// TwinCAT 3 PLC project kittingDeca
// ProgramVersion: 3.1.4023.0
// libraries:
//   Tc2_DataExchange, * (Beckhoff Automation GmbH)
//   Tc2_EtherCAT, * (Beckhoff Automation GmbH)
//   Tc2_MC2, * (Beckhoff Automation GmbH)
//   Tc2_SerialCom, * (Beckhoff Automation GmbH)
//   Tc2_Standard, * (Beckhoff Automation GmbH)
//   Tc2_System, * (Beckhoff Automation GmbH)
//   Tc2_Utilities, * (Beckhoff Automation GmbH)
//   Tc3_Module, * (Beckhoff Automation GmbH)
//   Tc3_PackML, * (Beckhoff Automation GmbH)
//   VisuDialogs, * (System)
//   VisuSymbols,3.5.10.0,System
// project tree:
//   DUTs/ user_defined_structure.TcDUT (not stored)
//   / GlobalTextList.TcGTLO, PlcTask.TcTTO, VISU_TASK.TcTTO, 视图管理器.TcVMO (not stored)
//   GVLs/ E_DOutputMode.TcDUT (not stored), E_State.TcDUT (not stored), ST_DIO.TcDUT (not stored), ST_IO.TcDUT (not stored), ST_IO_16.TcDUT (not stored), ST_IO_16_int.TcDUT (not stored)
//   GVLs/kitting deca/axis/ AxisHMI_Ex.TcVIS, E_HomingSteps.TcDUT (not stored), FB_MotionAxis_MC.TcPOU, MC_HomeAxis.TcPOU (not stored), ST_MotionAxis_MC.TcDUT
//   GVLs/kitting deca/ DigitalInputStatus.TcDUT (not stored), E_CMD_ConverterMotor.TcDUT, FB_Converter.TcPOU, FB_DigitalInput.TcPOU (not stored), FB_do.TcPOU (not stored), FB_PhotoSensor.TcPOU (not stored), FB_valve.TcPOU, Roller.TcDUT (not stored), Sensor.TcDUT (not stored), ST_Converter.TcDUT, ST_heightDetection.TcDUT, Valve.TcDUT (not stored)
//   GVLs/kitting deca/fixture rotation/ fixtureRotation_Module.TcDUT
//   GVLs/kitting deca/lateral conveyor/ BeltOut.TcDUT, Lateral.TcDUT, LateralBuf_Module.TcDUT, Roller_LC.TcDUT, LateralRecy_Module.TcDUT
//   GVLs/kitting deca/measuring/ ST_byte.TcDUT (not stored), ST_IO_byte.TcDUT (not stored)
//   GVLs/kitting deca/picking module/ Belt.TcDUT, Buffer.TcDUT (not stored), Inner_conveyor.TcDUT, PM_others.TcDUT (not stored), Outter_coveyor.TcDUT (not stored), Picking_Module.TcDUT (not stored), RFID.TcDUT (not stored)
//   GVLs/kitting deca/replenishment module/ arLiftAxis.TcDUT (not stored), Infeed.TcDUT (not stored), Lift.TcDUT (not stored), Outfeed.TcDUT (not stored), Replenishment_Module.TcDUT (not stored)
//   POUs/bagmachines/ AdsArr.TcDUT, BagCmd.TcDUT, BagDetectionCmd.TcDUT, BagDetectionStatus.TcDUT, BagHeightStatus.TcDUT, BagHolderStatus.TcDUT, BagMachineStatus.TcDUT, BagStatus.TcDUT, E_HeightDetection.TcDUT, FB_BagCloser.TcPOU, FB_BagCompactor.TcPOU, FB_BagOpener.TcPOU, fb_interface_bagmachine.TcPOU
//   POUs/ E_RemIndex.TcDUT (not stored), FB_axisCtrl.TcPOU, FB_heightDetection.TcPOU, FB_lbIOmapping.TcPOU, FB_frIOmapping.TcPOU, FB_remAxisMapping.TcPOU, FB_pmAxisMapping.TcPOU, FB_remIOmapping.TcPOU (not stored), FB_lcIOmapping.TcPOU, FB_rmIOmapping.TcPOU, G_HMI.TcGVL, GVL.TcGVL, G_IO.TcGVL, MAIN.TcPOU, ST_axisCtrl.TcDUT (not stored), ST_Color.TcDUT (not stored)
//   VISUs/ OtherList.TcVIS, visu_LC.TcVIS, visu_FR.TcVIS, visu_LB.TcVIS, visu_PM.TcVIS (not stored), visu_Others.TcVIS, visu_ReM.TcVIS, visu_MLC.TcVIS, visu_main.TcVIS, ReMList.TcVIS (not stored), PMList.TcVIS, v_byte.TcVIS (not stored), v_IO_FR.TcVIS, v_IO_fixtureClamp.TcVIS, v_IO_ReM.TcVIS (not stored), v_IO_LC.TcVIS, v_LB.TcVIS, v_rem_0.TcVIS, v_pm_0.TcVIS, v_rem_1.TcVIS
// real-time tasks:
//   TASK PlcTask: cycle T#2ms, priority 12, ADS port 350
//   TASK VISU_TASK: cycle T#200000us, priority 16, ADS port 351
// motion (NC):
//   TASK NC-Task 1 SAF: cycle T#4ms, priority 6, ADS port 501
//   TASK NC-Task 1 SVB: cycle T#10ms, priority 10, ADS port 511
//   AXIS rem0_Lift0 (id 4)
//     Dynamic: Acceleration=15000, Deceleration=15000, Jerk=150000
//     Velo: Maximum=3000
//     OtherSettings: AllowMotionCmdToSlave=true
//     encoder EncType=19
//       EncPara: ScaleFactorNumerator=5, ScaleFactorDenominator=262144, Inverse=true, MaxCount=#xffffffff
//         Inc: RefSoftSyncMask=#x00040000
//     drive DrvType=16
//       DrvPara: Inverse=true, MaxCount=#xffffffff, DriveControlDWord=#x00020100
//         Analog: VeloReferenz=500, TorqueSetpointScale=10, ScaleFactorActTorque=0.1
//         TimeComp: TaskDelayCycles=1
//     controller CtrType=1
//       CtrPara: PriorControlFactor=1
//         PosDiffControl: Range=30
//         Observer: BandWidth=20
//   AXIS rem0_Lift1 (id 5)
//     Dynamic: Acceleration=15000, Deceleration=15000, Jerk=150000
//     Velo: Maximum=3000
//     OtherSettings: AllowMotionCmdToSlave=true
//     encoder EncType=19
//       EncPara: ScaleFactorNumerator=5, ScaleFactorDenominator=262144, Inverse=true, MaxCount=#xffffffff
//         Inc: RefSoftSyncMask=#x00040000
//     drive DrvType=16
//       DrvPara: Inverse=true, MaxCount=#xffffffff, DriveControlDWord=#x00020100
//         Analog: VeloReferenz=500, TorqueSetpointScale=10, ScaleFactorActTorque=0.1
//         TimeComp: TaskDelayCycles=1
//     controller CtrType=1
//       CtrPara: PriorControlFactor=1
//         PosDiffControl: Range=30
//         Observer: BandWidth=20
//   AXIS rem1_Lift0 (id 1)
//     Dynamic: Acceleration=15000, Deceleration=15000, Jerk=150000
//     Velo: Maximum=3000
//     OtherSettings: AllowMotionCmdToSlave=true
//     encoder EncType=19
//       EncPara: ScaleFactorNumerator=5, ScaleFactorDenominator=262144, Inverse=true, MaxCount=#xffffffff
//         Inc: RefSoftSyncMask=#x00040000
//     drive DrvType=16
//       DrvPara: Inverse=true, MaxCount=#xffffffff, DriveControlDWord=#x00020100
//         Analog: VeloReferenz=500, TorqueSetpointScale=10, ScaleFactorActTorque=0.1
//         TimeComp: TaskDelayCycles=1
//     controller CtrType=1
//       CtrPara: PriorControlFactor=1
//         PosDiffControl: Range=30
//         Observer: BandWidth=20
//   AXIS rem1_Lift1 (id 2)
//     Dynamic: Acceleration=15000, Deceleration=15000, Jerk=150000
//     Velo: Maximum=3000
//     OtherSettings: AllowMotionCmdToSlave=true
//     encoder EncType=19
//       EncPara: ScaleFactorNumerator=5, ScaleFactorDenominator=262144, Inverse=true, MaxCount=#xffffffff
//         Inc: RefSoftSyncMask=#x00040000
//     drive DrvType=16
//       DrvPara: Inverse=true, MaxCount=#xffffffff, DriveControlDWord=#x00020100
//         Analog: VeloReferenz=500, TorqueSetpointScale=10, ScaleFactorActTorque=0.1
//         TimeComp: TaskDelayCycles=1
//     controller CtrType=1
//       CtrPara: PriorControlFactor=1
//         PosDiffControl: Range=30
//         Observer: BandWidth=20
//   AXIS rem2_Lift0 (id 9)
//     Dynamic: Acceleration=15000, Deceleration=15000, Jerk=150000
//     Velo: Maximum=3000
//     OtherSettings: AllowMotionCmdToSlave=true
//     encoder EncType=19
//       EncPara: ScaleFactorNumerator=5, ScaleFactorDenominator=262144, Inverse=true, MaxCount=#xffffffff
//         Inc: RefSoftSyncMask=#x00040000
//     drive DrvType=16
//       DrvPara: Inverse=true, MaxCount=#xffffffff, DriveControlDWord=#x00020100
//         Analog: VeloReferenz=500, TorqueSetpointScale=10, ScaleFactorActTorque=0.1
//         TimeComp: TaskDelayCycles=1
//     controller CtrType=1
//       CtrPara: PriorControlFactor=1
//         PosDiffControl: Range=30
//         Observer: BandWidth=20
//   AXIS rem2_Lift1 (id 10)
//     Dynamic: Acceleration=15000, Deceleration=15000, Jerk=150000
//     Velo: Maximum=3000
//     OtherSettings: AllowMotionCmdToSlave=true
//     encoder EncType=19
//       EncPara: ScaleFactorNumerator=5, ScaleFactorDenominator=262144, Inverse=true, MaxCount=#xffffffff
//         Inc: RefSoftSyncMask=#x00040000
//     drive DrvType=16
//       DrvPara: Inverse=true, MaxCount=#xffffffff, DriveControlDWord=#x00020100
//         Analog: VeloReferenz=500, TorqueSetpointScale=10, ScaleFactorActTorque=0.1
//         TimeComp: TaskDelayCycles=1
//     controller CtrType=1
//       CtrPara: PriorControlFactor=1
//         PosDiffControl: Range=30
//         Observer: BandWidth=20
//   AXIS rem3_Lift0 (id 11)
//     Dynamic: Acceleration=15000, Deceleration=15000, Jerk=150000
//     Velo: Maximum=3000
//     OtherSettings: AllowMotionCmdToSlave=true
//     encoder EncType=19
//       EncPara: ScaleFactorNumerator=5, ScaleFactorDenominator=262144, Inverse=true, MaxCount=#xffffffff
//         Inc: RefSoftSyncMask=#x00040000
//     drive DrvType=16
//       DrvPara: Inverse=true, MaxCount=#xffffffff, DriveControlDWord=#x00020100
//         Analog: VeloReferenz=500, TorqueSetpointScale=10, ScaleFactorActTorque=0.1
//         TimeComp: TaskDelayCycles=1
//     controller CtrType=1
//       CtrPara: PriorControlFactor=1
//         PosDiffControl: Range=30
//         Observer: BandWidth=20
//   AXIS rem3_Lift1 (id 12)
//     Dynamic: Acceleration=15000, Deceleration=15000, Jerk=150000
//     Velo: Maximum=3000
//     OtherSettings: AllowMotionCmdToSlave=true
//     encoder EncType=19
//       EncPara: ScaleFactorNumerator=5, ScaleFactorDenominator=262144, Inverse=true, MaxCount=#xffffffff
//         Inc: RefSoftSyncMask=#x00040000
//     drive DrvType=16
//       DrvPara: Inverse=true, MaxCount=#xffffffff, DriveControlDWord=#x00020100
//         Analog: VeloReferenz=500, TorqueSetpointScale=10, ScaleFactorActTorque=0.1
//         TimeComp: TaskDelayCycles=1
//     controller CtrType=1
//       CtrPara: PriorControlFactor=1
//         PosDiffControl: Range=30
//         Observer: BandWidth=20
//   AXIS rem4_Lift0 (id 17)
//     Dynamic: Acceleration=15000, Deceleration=15000, Jerk=150000
//     Velo: Maximum=3000
//     OtherSettings: AllowMotionCmdToSlave=true
//     encoder EncType=19
//       EncPara: ScaleFactorNumerator=5, ScaleFactorDenominator=262144, Inverse=true, MaxCount=#xffffffff
//         Inc: RefSoftSyncMask=#x00040000
//     drive DrvType=16
//       DrvPara: Inverse=true, MaxCount=#xffffffff, DriveControlDWord=#x00020100
//         Analog: VeloReferenz=500, TorqueSetpointScale=10, ScaleFactorActTorque=0.1
//         TimeComp: TaskDelayCycles=1
//     controller CtrType=1
//       CtrPara: PriorControlFactor=1
//         PosDiffControl: Range=30
//         Observer: BandWidth=20
//   AXIS rem4_Lift1 (id 18)
//     Dynamic: Acceleration=15000, Deceleration=15000, Jerk=150000
//     Velo: Maximum=3000
//     OtherSettings: AllowMotionCmdToSlave=true
//     encoder EncType=19
//       EncPara: ScaleFactorNumerator=5, ScaleFactorDenominator=262144, Inverse=true, MaxCount=#xffffffff
//         Inc: RefSoftSyncMask=#x00040000
//     drive DrvType=16
//       DrvPara: Inverse=true, MaxCount=#xffffffff, DriveControlDWord=#x00020100
//         Analog: VeloReferenz=500, TorqueSetpointScale=10, ScaleFactorActTorque=0.1
//         TimeComp: TaskDelayCycles=1
//     controller CtrType=1
//       CtrPara: PriorControlFactor=1
//         PosDiffControl: Range=30
//         Observer: BandWidth=20
//   AXIS rem5_Lift0 (id 19)
//     Dynamic: Acceleration=15000, Deceleration=15000, Jerk=150000
//     Velo: Maximum=3000
//     OtherSettings: AllowMotionCmdToSlave=true
//     encoder EncType=19
//       EncPara: ScaleFactorNumerator=5, ScaleFactorDenominator=262144, Inverse=true, MaxCount=#xffffffff
//         Inc: RefSoftSyncMask=#x00040000
//     drive DrvType=16
//       DrvPara: Inverse=true, MaxCount=#xffffffff, DriveControlDWord=#x00020100
//         Analog: VeloReferenz=500, TorqueSetpointScale=10, ScaleFactorActTorque=0.1
//         TimeComp: TaskDelayCycles=1
//     controller CtrType=1
//       CtrPara: PriorControlFactor=1
//         PosDiffControl: Range=30
//         Observer: BandWidth=20
//   AXIS rem5_Lift1 (id 20)
//     Dynamic: Acceleration=15000, Deceleration=15000, Jerk=150000
//     Velo: Maximum=3000
//     OtherSettings: AllowMotionCmdToSlave=true
//     encoder EncType=19
//       EncPara: ScaleFactorNumerator=5, ScaleFactorDenominator=262144, Inverse=true, MaxCount=#xffffffff
//         Inc: RefSoftSyncMask=#x00040000
//     drive DrvType=16
//       DrvPara: Inverse=true, MaxCount=#xffffffff, DriveControlDWord=#x00020100
//         Analog: VeloReferenz=500, TorqueSetpointScale=10, ScaleFactorActTorque=0.1
//         TimeComp: TaskDelayCycles=1
//     controller CtrType=1
//       CtrPara: PriorControlFactor=1
//         PosDiffControl: Range=30
//         Observer: BandWidth=20
//   AXIS rem6_Lift0 (id 25)
//     Dynamic: Acceleration=15000, Deceleration=15000, Jerk=150000
//     Velo: Maximum=3000
//     OtherSettings: AllowMotionCmdToSlave=true
//     encoder EncType=19
//       EncPara: ScaleFactorNumerator=5, ScaleFactorDenominator=262144, Inverse=true, MaxCount=#xffffffff
//         Inc: RefSoftSyncMask=#x00040000
//     drive DrvType=16
//       DrvPara: Inverse=true, MaxCount=#xffffffff, DriveControlDWord=#x00020100
//         Analog: VeloReferenz=500, TorqueSetpointScale=10, ScaleFactorActTorque=0.1
//         TimeComp: TaskDelayCycles=1
//     controller CtrType=1
//       CtrPara: PriorControlFactor=1
//         PosDiffControl: Range=30
//         Observer: BandWidth=20
//   AXIS rem6_Lift1 (id 26)
//     Dynamic: Acceleration=15000, Deceleration=15000, Jerk=150000
//     Velo: Maximum=3000
//     OtherSettings: AllowMotionCmdToSlave=true
//     encoder EncType=19
//       EncPara: ScaleFactorNumerator=5, ScaleFactorDenominator=262144, Inverse=true, MaxCount=#xffffffff
//         Inc: RefSoftSyncMask=#x00040000
//     drive DrvType=16
//       DrvPara: Inverse=true, MaxCount=#xffffffff, DriveControlDWord=#x00020100
//         Analog: VeloReferenz=500, TorqueSetpointScale=10, ScaleFactorActTorque=0.1
//         TimeComp: TaskDelayCycles=1
//     controller CtrType=1
//       CtrPara: PriorControlFactor=1
//         PosDiffControl: Range=30
//         Observer: BandWidth=20
//   AXIS rem7_Lift0 (id 27)
//     Dynamic: Acceleration=15000, Deceleration=15000, Jerk=150000
//     Velo: Maximum=3000
//     OtherSettings: AllowMotionCmdToSlave=true
//     encoder EncType=19
//       EncPara: ScaleFactorNumerator=5, ScaleFactorDenominator=262144, Inverse=true, MaxCount=#xffffffff
//         Inc: RefSoftSyncMask=#x00040000
//     drive DrvType=16
//       DrvPara: Inverse=true, MaxCount=#xffffffff, DriveControlDWord=#x00020100
//         Analog: VeloReferenz=500, TorqueSetpointScale=10, ScaleFactorActTorque=0.1
//         TimeComp: TaskDelayCycles=1
//     controller CtrType=1
//       CtrPara: PriorControlFactor=1
//         PosDiffControl: Range=30
//         Observer: BandWidth=20
//   AXIS rem7_Lift1 (id 28)
//     Dynamic: Acceleration=15000, Deceleration=15000, Jerk=150000
//     Velo: Maximum=3000
//     OtherSettings: AllowMotionCmdToSlave=true
//     encoder EncType=19
//       EncPara: ScaleFactorNumerator=5, ScaleFactorDenominator=262144, Inverse=true, MaxCount=#xffffffff
//         Inc: RefSoftSyncMask=#x00040000
//     drive DrvType=16
//       DrvPara: Inverse=true, MaxCount=#xffffffff, DriveControlDWord=#x00020100
//         Analog: VeloReferenz=500, TorqueSetpointScale=10, ScaleFactorActTorque=0.1
//         TimeComp: TaskDelayCycles=1
//     controller CtrType=1
//       CtrPara: PriorControlFactor=1
//         PosDiffControl: Range=30
//         Observer: BandWidth=20
//   AXIS rem8_Lift0 (id 33)
//     Dynamic: Acceleration=15000, Deceleration=15000, Jerk=150000
//     Velo: Maximum=3000
//     OtherSettings: AllowMotionCmdToSlave=true
//     encoder EncType=19
//       EncPara: ScaleFactorNumerator=5, ScaleFactorDenominator=262144, Inverse=true, MaxCount=#xffffffff
//         Inc: RefSoftSyncMask=#x00040000
//     drive DrvType=16
//       DrvPara: Inverse=true, MaxCount=#xffffffff, DriveControlDWord=#x00020100
//         Analog: VeloReferenz=500, TorqueSetpointScale=10, ScaleFactorActTorque=0.1
//         TimeComp: TaskDelayCycles=1
//     controller CtrType=1
//       CtrPara: PriorControlFactor=1
//         PosDiffControl: Range=30
//         Observer: BandWidth=20
//   AXIS rem8_Lift1 (id 34)
//     Dynamic: Acceleration=15000, Deceleration=15000, Jerk=150000
//     Velo: Maximum=3000
//     OtherSettings: AllowMotionCmdToSlave=true
//     encoder EncType=19
//       EncPara: ScaleFactorNumerator=5, ScaleFactorDenominator=262144, Inverse=true, MaxCount=#xffffffff
//         Inc: RefSoftSyncMask=#x00040000
//     drive DrvType=16
//       DrvPara: Inverse=true, MaxCount=#xffffffff, DriveControlDWord=#x00020100
//         Analog: VeloReferenz=500, TorqueSetpointScale=10, ScaleFactorActTorque=0.1
//         TimeComp: TaskDelayCycles=1
//     controller CtrType=1
//       CtrPara: PriorControlFactor=1
//         PosDiffControl: Range=30
//         Observer: BandWidth=20
//   AXIS rem9_Lift0 (id 35)
//     Dynamic: Acceleration=15000, Deceleration=15000, Jerk=150000
//     Velo: Maximum=3000
//     OtherSettings: AllowMotionCmdToSlave=true
//     encoder EncType=19
//       EncPara: ScaleFactorNumerator=5, ScaleFactorDenominator=262144, Inverse=true, MaxCount=#xffffffff
//         Inc: RefSoftSyncMask=#x00040000
//     drive DrvType=16
//       DrvPara: Inverse=true, MaxCount=#xffffffff, DriveControlDWord=#x00020100
//         Analog: VeloReferenz=500, TorqueSetpointScale=10, ScaleFactorActTorque=0.1
//         TimeComp: TaskDelayCycles=1
//     controller CtrType=1
//       CtrPara: PriorControlFactor=1
//         PosDiffControl: Range=30
//         Observer: BandWidth=20
//   AXIS rem9_Lift1 (id 36)
//     Dynamic: Acceleration=15000, Deceleration=15000, Jerk=150000
//     Velo: Maximum=3000
//     OtherSettings: AllowMotionCmdToSlave=true
//     encoder EncType=19
//       EncPara: ScaleFactorNumerator=5, ScaleFactorDenominator=262144, Inverse=true, MaxCount=#xffffffff
//         Inc: RefSoftSyncMask=#x00040000
//     drive DrvType=16
//       DrvPara: Inverse=true, MaxCount=#xffffffff, DriveControlDWord=#x00020100
//         Analog: VeloReferenz=500, TorqueSetpointScale=10, ScaleFactorActTorque=0.1
//         TimeComp: TaskDelayCycles=1
//     controller CtrType=1
//       CtrPara: PriorControlFactor=1
//         PosDiffControl: Range=30
//         Observer: BandWidth=20
//   AXIS pm0_buf0 (id 3)
//     Dynamic: Acceleration=15000, Deceleration=15000, Jerk=150000
//     Velo: Maximum=3000
//     OtherSettings: AllowMotionCmdToSlave=true
//     encoder EncType=19
//       EncPara: ScaleFactorNumerator=20.84, ScaleFactorDenominator=262144, MaxCount=#xffffffff
//         Inc: RefSoftSyncMask=#x00040000
//     drive DrvType=16
//       DrvPara: MaxCount=#xffffffff, DriveControlDWord=#x00020100
//         Analog: VeloReferenz=500, TorqueSetpointScale=10, ScaleFactorActTorque=0.1
//         TimeComp: TaskDelayCycles=1
//     controller CtrType=1
//       CtrPara: PriorControlFactor=1
//         PosDiffControl: Range=30
//         Observer: BandWidth=20
//   AXIS pm0_buf1 (id 6)
//     Dynamic: Acceleration=15000, Deceleration=15000, Jerk=150000
//     Velo: Maximum=3000
//     OtherSettings: AllowMotionCmdToSlave=true
//     encoder EncType=19
//       EncPara: ScaleFactorNumerator=20.84, ScaleFactorDenominator=262144, MaxCount=#xffffffff
//         Inc: RefSoftSyncMask=#x00040000
//     drive DrvType=16
//       DrvPara: MaxCount=#xffffffff, DriveControlDWord=#x00020100
//         Analog: VeloReferenz=500, TorqueSetpointScale=10, ScaleFactorActTorque=0.1
//         TimeComp: TaskDelayCycles=1
//     controller CtrType=1
//       CtrPara: PriorControlFactor=1
//         PosDiffControl: Range=30
//         Observer: BandWidth=20
//   AXIS pm1_buf0 (id 7)
//     Dynamic: Acceleration=15000, Deceleration=15000, Jerk=150000
//     Velo: Maximum=3000
//     OtherSettings: AllowMotionCmdToSlave=true
//     encoder EncType=19
//       EncPara: ScaleFactorNumerator=20.84, ScaleFactorDenominator=262144, MaxCount=#xffffffff
//         Inc: RefSoftSyncMask=#x00040000
//     drive DrvType=16
//       DrvPara: MaxCount=#xffffffff, DriveControlDWord=#x00020100
//         Analog: VeloReferenz=500, TorqueSetpointScale=10, ScaleFactorActTorque=0.1
//         TimeComp: TaskDelayCycles=1
//     controller CtrType=1
//       CtrPara: PriorControlFactor=1
//         PosDiffControl: Range=30
//         Observer: BandWidth=20
//   AXIS pm1_buf1 (id 8)
//     Dynamic: Acceleration=15000, Deceleration=15000, Jerk=150000
//     Velo: Maximum=3000
//     OtherSettings: AllowMotionCmdToSlave=true
//     encoder EncType=19
//       EncPara: ScaleFactorNumerator=20.84, ScaleFactorDenominator=262144, MaxCount=#xffffffff
//         Inc: RefSoftSyncMask=#x00040000
//     drive DrvType=16
//       DrvPara: MaxCount=#xffffffff, DriveControlDWord=#x00020100
//         Analog: VeloReferenz=500, TorqueSetpointScale=10, ScaleFactorActTorque=0.1
//         TimeComp: TaskDelayCycles=1
//     controller CtrType=1
//       CtrPara: PriorControlFactor=1
//         PosDiffControl: Range=30
//         Observer: BandWidth=20
//   AXIS pm2_buf0 (id 13)
//     Dynamic: Acceleration=15000, Deceleration=15000, Jerk=150000
//     Velo: Maximum=3000
//     OtherSettings: AllowMotionCmdToSlave=true
//     encoder EncType=19
//       EncPara: ScaleFactorNumerator=20.84, ScaleFactorDenominator=262144, MaxCount=#xffffffff
//         Inc: RefSoftSyncMask=#x00040000
//     drive DrvType=16
//       DrvPara: MaxCount=#xffffffff, DriveControlDWord=#x00020100
//         Analog: VeloReferenz=500, TorqueSetpointScale=10, ScaleFactorActTorque=0.1
//         TimeComp: TaskDelayCycles=1
//     controller CtrType=1
//       CtrPara: PriorControlFactor=1
//         PosDiffControl: Range=30
//         Observer: BandWidth=20
//   AXIS pm2_buf1 (id 14)
//     Dynamic: Acceleration=15000, Deceleration=15000, Jerk=150000
//     Velo: Maximum=3000
//     OtherSettings: AllowMotionCmdToSlave=true
//     encoder EncType=19
//       EncPara: ScaleFactorNumerator=20.84, ScaleFactorDenominator=262144, MaxCount=#xffffffff
//         Inc: RefSoftSyncMask=#x00040000
//     drive DrvType=16
//       DrvPara: MaxCount=#xffffffff, DriveControlDWord=#x00020100
//         Analog: VeloReferenz=500, TorqueSetpointScale=10, ScaleFactorActTorque=0.1
//         TimeComp: TaskDelayCycles=1
//     controller CtrType=1
//       CtrPara: PriorControlFactor=1
//         PosDiffControl: Range=30
//         Observer: BandWidth=20
//   AXIS pm3_buf0 (id 15)
//     Dynamic: Acceleration=15000, Deceleration=15000, Jerk=150000
//     Velo: Maximum=3000
//     OtherSettings: AllowMotionCmdToSlave=true
//     encoder EncType=19
//       EncPara: ScaleFactorNumerator=20.84, ScaleFactorDenominator=262144, MaxCount=#xffffffff
//         Inc: RefSoftSyncMask=#x00040000
//     drive DrvType=16
//       DrvPara: MaxCount=#xffffffff, DriveControlDWord=#x00020100
//         Analog: VeloReferenz=500, TorqueSetpointScale=10, ScaleFactorActTorque=0.1
//         TimeComp: TaskDelayCycles=1
//     controller CtrType=1
//       CtrPara: PriorControlFactor=1
//         PosDiffControl: Range=30
//         Observer: BandWidth=20
//   AXIS pm3_buf1 (id 16)
//     Dynamic: Acceleration=15000, Deceleration=15000, Jerk=150000
//     Velo: Maximum=3000
//     OtherSettings: AllowMotionCmdToSlave=true
//     encoder EncType=19
//       EncPara: ScaleFactorNumerator=20.84, ScaleFactorDenominator=262144, MaxCount=#xffffffff
//         Inc: RefSoftSyncMask=#x00040000
//     drive DrvType=16
//       DrvPara: MaxCount=#xffffffff, DriveControlDWord=#x00020100
//         Analog: VeloReferenz=500, TorqueSetpointScale=10, ScaleFactorActTorque=0.1
//         TimeComp: TaskDelayCycles=1
//     controller CtrType=1
//       CtrPara: PriorControlFactor=1
//         PosDiffControl: Range=30
//         Observer: BandWidth=20
//   AXIS pm4_buf0 (id 21)
//     Dynamic: Acceleration=15000, Deceleration=15000, Jerk=150000
//     Velo: Maximum=3000
//     OtherSettings: AllowMotionCmdToSlave=true
//     encoder EncType=19
//       EncPara: ScaleFactorNumerator=20.84, ScaleFactorDenominator=262144, MaxCount=#xffffffff
//         Inc: RefSoftSyncMask=#x00040000
//     drive DrvType=16
//       DrvPara: MaxCount=#xffffffff, DriveControlDWord=#x00020100
//         Analog: VeloReferenz=500, TorqueSetpointScale=10, ScaleFactorActTorque=0.1
//         TimeComp: TaskDelayCycles=1
//     controller CtrType=1
//       CtrPara: PriorControlFactor=1
//         PosDiffControl: Range=30
//         Observer: BandWidth=20
//   AXIS pm4_buf1 (id 22)
//     Dynamic: Acceleration=15000, Deceleration=15000, Jerk=150000
//     Velo: Maximum=3000
//     OtherSettings: AllowMotionCmdToSlave=true
//     encoder EncType=19
//       EncPara: ScaleFactorNumerator=20.84, ScaleFactorDenominator=262144, MaxCount=#xffffffff
//         Inc: RefSoftSyncMask=#x00040000
//     drive DrvType=16
//       DrvPara: MaxCount=#xffffffff, DriveControlDWord=#x00020100
//         Analog: VeloReferenz=500, TorqueSetpointScale=10, ScaleFactorActTorque=0.1
//         TimeComp: TaskDelayCycles=1
//     controller CtrType=1
//       CtrPara: PriorControlFactor=1
//         PosDiffControl: Range=30
//         Observer: BandWidth=20
//   AXIS pm5_buf0 (id 23)
//     Dynamic: Acceleration=15000, Deceleration=15000, Jerk=150000
//     Velo: Maximum=3000
//     OtherSettings: AllowMotionCmdToSlave=true
//     encoder EncType=19
//       EncPara: ScaleFactorNumerator=20.84, ScaleFactorDenominator=262144, MaxCount=#xffffffff
//         Inc: RefSoftSyncMask=#x00040000
//     drive DrvType=16
//       DrvPara: MaxCount=#xffffffff, DriveControlDWord=#x00020100
//         Analog: VeloReferenz=500, TorqueSetpointScale=10, ScaleFactorActTorque=0.1
//         TimeComp: TaskDelayCycles=1
//     controller CtrType=1
//       CtrPara: PriorControlFactor=1
//         PosDiffControl: Range=30
//         Observer: BandWidth=20
//   AXIS pm5_buf1 (id 24)
//     Dynamic: Acceleration=15000, Deceleration=15000, Jerk=150000
//     Velo: Maximum=3000
//     OtherSettings: AllowMotionCmdToSlave=true
//     encoder EncType=19
//       EncPara: ScaleFactorNumerator=20.84, ScaleFactorDenominator=262144, MaxCount=#xffffffff
//         Inc: RefSoftSyncMask=#x00040000
//     drive DrvType=16
//       DrvPara: MaxCount=#xffffffff, DriveControlDWord=#x00020100
//         Analog: VeloReferenz=500, TorqueSetpointScale=10, ScaleFactorActTorque=0.1
//         TimeComp: TaskDelayCycles=1
//     controller CtrType=1
//       CtrPara: PriorControlFactor=1
//         PosDiffControl: Range=30
//         Observer: BandWidth=20
//   AXIS pm6_buf0 (id 29)
//     Dynamic: Acceleration=15000, Deceleration=15000, Jerk=150000
//     Velo: Maximum=3000
//     OtherSettings: AllowMotionCmdToSlave=true
//     encoder EncType=19
//       EncPara: ScaleFactorNumerator=20.84, ScaleFactorDenominator=262144, MaxCount=#xffffffff
//         Inc: RefSoftSyncMask=#x00040000
//     drive DrvType=16
//       DrvPara: MaxCount=#xffffffff, DriveControlDWord=#x00020100
//         Analog: VeloReferenz=500, TorqueSetpointScale=10, ScaleFactorActTorque=0.1
//         TimeComp: TaskDelayCycles=1
//     controller CtrType=1
//       CtrPara: PriorControlFactor=1
//         PosDiffControl: Range=30
//         Observer: BandWidth=20
//   AXIS pm6_buf1 (id 30)
//     Dynamic: Acceleration=15000, Deceleration=15000, Jerk=150000
//     Velo: Maximum=3000
//     OtherSettings: AllowMotionCmdToSlave=true
//     encoder EncType=19
//       EncPara: ScaleFactorNumerator=20.84, ScaleFactorDenominator=262144, MaxCount=#xffffffff
//         Inc: RefSoftSyncMask=#x00040000
//     drive DrvType=16
//       DrvPara: MaxCount=#xffffffff, DriveControlDWord=#x00020100
//         Analog: VeloReferenz=500, TorqueSetpointScale=10, ScaleFactorActTorque=0.1
//         TimeComp: TaskDelayCycles=1
//     controller CtrType=1
//       CtrPara: PriorControlFactor=1
//         PosDiffControl: Range=30
//         Observer: BandWidth=20
//   AXIS pm7_buf0 (id 31)
//     Dynamic: Acceleration=15000, Deceleration=15000, Jerk=150000
//     Velo: Maximum=3000
//     OtherSettings: AllowMotionCmdToSlave=true
//     encoder EncType=19
//       EncPara: ScaleFactorNumerator=20.84, ScaleFactorDenominator=262144, MaxCount=#xffffffff
//         Inc: RefSoftSyncMask=#x00040000
//     drive DrvType=16
//       DrvPara: MaxCount=#xffffffff, DriveControlDWord=#x00020100
//         Analog: VeloReferenz=500, TorqueSetpointScale=10, ScaleFactorActTorque=0.1
//         TimeComp: TaskDelayCycles=1
//     controller CtrType=1
//       CtrPara: PriorControlFactor=1
//         PosDiffControl: Range=30
//         Observer: BandWidth=20
//   AXIS pm7_buf1 (id 32)
//     Dynamic: Acceleration=15000, Deceleration=15000, Jerk=150000
//     Velo: Maximum=3000
//     OtherSettings: AllowMotionCmdToSlave=true
//     encoder EncType=19
//       EncPara: ScaleFactorNumerator=20.84, ScaleFactorDenominator=262144, MaxCount=#xffffffff
//         Inc: RefSoftSyncMask=#x00040000
//     drive DrvType=16
//       DrvPara: MaxCount=#xffffffff, DriveControlDWord=#x00020100
//         Analog: VeloReferenz=500, TorqueSetpointScale=10, ScaleFactorActTorque=0.1
//         TimeComp: TaskDelayCycles=1
//     controller CtrType=1
//       CtrPara: PriorControlFactor=1
//         PosDiffControl: Range=30
//         Observer: BandWidth=20
//   AXIS pm8_buf0 (id 37)
//     Dynamic: Acceleration=15000, Deceleration=15000, Jerk=150000
//     Velo: Maximum=3000
//     OtherSettings: AllowMotionCmdToSlave=true
//     encoder EncType=19
//       EncPara: ScaleFactorNumerator=20.84, ScaleFactorDenominator=262144, MaxCount=#xffffffff
//         Inc: RefSoftSyncMask=#x00040000
//     drive DrvType=16
//       DrvPara: MaxCount=#xffffffff, DriveControlDWord=#x00020100
//         Analog: VeloReferenz=500, TorqueSetpointScale=10, ScaleFactorActTorque=0.1
//         TimeComp: TaskDelayCycles=1
//     controller CtrType=1
//       CtrPara: PriorControlFactor=1
//         PosDiffControl: Range=30
//         Observer: BandWidth=20
//   AXIS pm8_buf1 (id 38)
//     Dynamic: Acceleration=15000, Deceleration=15000, Jerk=150000
//     Velo: Maximum=3000
//     OtherSettings: AllowMotionCmdToSlave=true
//     encoder EncType=19
//       EncPara: ScaleFactorNumerator=20.84, ScaleFactorDenominator=262144, MaxCount=#xffffffff
//         Inc: RefSoftSyncMask=#x00040000
//     drive DrvType=16
//       DrvPara: MaxCount=#xffffffff, DriveControlDWord=#x00020100
//         Analog: VeloReferenz=500, TorqueSetpointScale=10, ScaleFactorActTorque=0.1
//         TimeComp: TaskDelayCycles=1
//     controller CtrType=1
//       CtrPara: PriorControlFactor=1
//         PosDiffControl: Range=30
//         Observer: BandWidth=20
//   AXIS pm9_buf0 (id 39)
//     Dynamic: Acceleration=15000, Deceleration=15000, Jerk=150000
//     Velo: Maximum=3000
//     OtherSettings: AllowMotionCmdToSlave=true
//     encoder EncType=19
//       EncPara: ScaleFactorNumerator=20.84, ScaleFactorDenominator=262144, MaxCount=#xffffffff
//         Inc: RefSoftSyncMask=#x00040000
//     drive DrvType=16
//       DrvPara: MaxCount=#xffffffff, DriveControlDWord=#x00020100
//         Analog: VeloReferenz=500, TorqueSetpointScale=10, ScaleFactorActTorque=0.1
//         TimeComp: TaskDelayCycles=1
//     controller CtrType=1
//       CtrPara: PriorControlFactor=1
//         PosDiffControl: Range=30
//         Observer: BandWidth=20
//   AXIS pm9_buf1 (id 40)
//     Dynamic: Acceleration=15000, Deceleration=15000, Jerk=150000
//     Velo: Maximum=3000
//     OtherSettings: AllowMotionCmdToSlave=true
//     encoder EncType=19
//       EncPara: ScaleFactorNumerator=20.84, ScaleFactorDenominator=262144, MaxCount=#xffffffff
//         Inc: RefSoftSyncMask=#x00040000
//     drive DrvType=16
//       DrvPara: MaxCount=#xffffffff, DriveControlDWord=#x00020100
//         Analog: VeloReferenz=500, TorqueSetpointScale=10, ScaleFactorActTorque=0.1
//         TimeComp: TaskDelayCycles=1
//     controller CtrType=1
//       CtrPara: PriorControlFactor=1
//         PosDiffControl: Range=30
//         Observer: BandWidth=20
//   AXIS fr0 (id 41)
//     Dynamic: Acceleration=15000, Deceleration=15000, Jerk=150000
//     Velo: Maximum=3000
//     OtherSettings: AllowMotionCmdToSlave=true
//     encoder EncType=19
//       EncPara: ScaleFactorNumerator=7.2, ScaleFactorDenominator=262144, MaxCount=#xffffffff
//         Inc: RefSoftSyncMask=#x00040000
//     drive DrvType=16
//       DrvPara: MaxCount=#xffffffff, DriveControlDWord=#x00020100
//         Analog: VeloReferenz=500, TorqueSetpointScale=10, ScaleFactorActTorque=0.1
//         TimeComp: TaskDelayCycles=1
//     controller CtrType=1
//       CtrPara: PriorControlFactor=1
//         PosDiffControl: Range=30
//         Observer: BandWidth=20
//   AXIS fr1 (id 42)
//     Dynamic: Acceleration=15000, Deceleration=15000, Jerk=150000
//     Velo: Maximum=3000
//     OtherSettings: AllowMotionCmdToSlave=true
//     encoder EncType=19
//       EncPara: ScaleFactorNumerator=7.2, ScaleFactorDenominator=262144, MaxCount=#xffffffff
//         Inc: RefSoftSyncMask=#x00040000
//     drive DrvType=16
//       DrvPara: MaxCount=#xffffffff, DriveControlDWord=#x00020100
//         Analog: VeloReferenz=500, TorqueSetpointScale=10, ScaleFactorActTorque=0.1
//         TimeComp: TaskDelayCycles=1
//     controller CtrType=1
//       CtrPara: PriorControlFactor=1
//         PosDiffControl: Range=30
//         Observer: BandWidth=20
//   AXIS lc0 (id 43)
//     Dynamic: Acceleration=15000, Deceleration=15000, Jerk=150000
//     Velo: Maximum=3000
//     OtherSettings: AllowMotionCmdToSlave=true
//     encoder EncType=19
//       EncPara: ScaleFactorNumerator=20, ScaleFactorDenominator=262144, MaxCount=#xffffffff
//         Inc: RefSoftSyncMask=#x00040000
//     drive DrvType=16
//       DrvPara: MaxCount=#xffffffff, DriveControlDWord=#x00020100
//         Analog: VeloReferenz=1000, TorqueSetpointScale=10, ScaleFactorActTorque=0.1
//         TimeComp: TaskDelayCycles=1
//     controller CtrType=1
//       CtrPara: PriorControlFactor=1
//         PosDiffControl: Range=30
//         Observer: BandWidth=20
//   AXIS lc1 (id 44)
//     Dynamic: Acceleration=15000, Deceleration=15000, Jerk=150000
//     Velo: Maximum=3000
//     OtherSettings: AllowMotionCmdToSlave=true
//     encoder EncType=19
//       EncPara: ScaleFactorNumerator=20, ScaleFactorDenominator=262144, MaxCount=#xffffffff
//         Inc: RefSoftSyncMask=#x00040000
//     drive DrvType=16
//       DrvPara: MaxCount=#xffffffff, DriveControlDWord=#x00020100
//         Analog: VeloReferenz=1000, TorqueSetpointScale=10, ScaleFactorActTorque=0.1
//         TimeComp: TaskDelayCycles=1
//     controller CtrType=1
//       CtrPara: PriorControlFactor=1
//         PosDiffControl: Range=30
//         Observer: BandWidth=20
// I/O:
//   DEVICE Device 1 (EtherCAT Automation Protocol), AmsNetId 192.168.11.159.2.1
//   DEVICE Device 2 (RT-Ethernet Adapter)
//   DEVICE rem_wf, AmsNetId 192.168.11.159.4.1
//     Box 1 (CU2508) [CU2508 Ethernet Port]
//     mcp_dio [GL20-RTU-ECT_1.3.5.0]
//       modules: Module 1 (GL20-1600END), Module 2 (GL20-0016ETP)
//     safetyPLC [Flexi Soft EtherCAT Gateway]
//     rem0_dio [GL20-RTU-ECT_1.3.5.0]
//       modules: DI0, DI1, DI2, DI3, DO0, DO1
//     rem0_Lift0 [SV630_1Axis_03713]
//     rem0_Lift1 [SV630_1Axis_03713]
//     rem0_valve [C2S-EC]
//       modules: Module 1 (C2S-EC-24B)
//     rem1_dio [GL20-RTU-ECT_1.3.5.0]
//       modules: DI4, DI5, DI6, DI7, DO4, DO5
//     rem1_Lift0 [SV630_1Axis_03713]
//     rem1_Lift1 [SV630_1Axis_03713]
//     rem1_valve [C2S-EC]
//       modules: Module 1 (C2S-EC-24B)
//     rem2_dio [GL20-RTU-ECT_1.3.5.0]
//       modules: DI8, DI9, DI10, DI11, DO8, DO9
//     rem2_Lift0 [SV630_1Axis_03713]
//     rem2_Lift1 [SV630_1Axis_03713]
//     rem2_valve [C2S-EC]
//       modules: Module 1 (C2S-EC-24B)
//     rem3_dio [GL20-RTU-ECT_1.3.5.0]
//       modules: DI12, DI13, DI14, DI15, DO12, DO13
//     rem3_Lift0 [SV630_1Axis_03713]
//     rem3_Lift1 [SV630_1Axis_03713]
//     rem3_valve [C2S-EC]
//       modules: Module 1 (C2S-EC-24B)
//     rem4_dio [GL20-RTU-ECT_1.3.5.0]
//       modules: DI0, DI1, DI2, DI3, DO0, DO1
//     rem4_Lift0 [SV630_1Axis_03713]
//     rem4_Lift1 [SV630_1Axis_03713]
//     rem4_valve [C2S-EC]
//       modules: Module 1 (C2S-EC-24B)
//     rem5_dio [GL20-RTU-ECT_1.3.5.0]
//       modules: DI0, DI1, DI2, DI3, DO0, DO1
//     rem5_Lift0 [SV630_1Axis_03713]
//     rem5_Lift1 [SV630_1Axis_03713]
//     rem5_valve [C2S-EC]
//       modules: Module 1 (C2S-EC-24B)
//     rem6_dio [GL20-RTU-ECT_1.3.5.0]
//       modules: DI0, DI1, DI2, DI3, DO0, DO1
//     rem6_Lift0 [SV630_1Axis_03713]
//     rem6_Lift1 [SV630_1Axis_03713]
//     rem6_valve [C2S-EC]
//       modules: Module 1 (C2S-EC-24B)
//     rem7_dio [GL20-RTU-ECT_1.3.5.0]
//       modules: DI0, DI1, DI2, DI3, DO0, DO1
//     rem7_Lift0 [SV630_1Axis_03713]
//     rem7_Lift1 [SV630_1Axis_03713]
//     rem7_valve [C2S-EC]
//       modules: Module 1 (C2S-EC-24B)
//     rem8_dio [GL20-RTU-ECT_1.3.5.0]
//       modules: DI0, DI1, DI2, DI3, DO0, DO1
//     rem8_Lift0 [SV630_1Axis_03713]
//     rem8_Lift1 [SV630_1Axis_03713]
//     rem8_valve [C2S-EC]
//       modules: Module 1 (C2S-EC-24B)
//     rem9_dio [GL20-RTU-ECT_1.3.5.0]
//       modules: DI0, DI1, DI2, DI3, DO0, DO1
//     rem9_Lift0 [SV630_1Axis_03713]
//     rem9_Lift1 [SV630_1Axis_03713]
//     rem9_valve [C2S-EC]
//       modules: Module 1 (C2S-EC-24B)
//     wf4_do [GL20-RTU-ECT_1.3.5.0]
//       modules: Module 1 (GL20-0016ETP), Module 2 (GL20-1600END)
//     wf3_do [GL20-RTU-ECT_1.3.5.0]
//       modules: Module 1 (GL20-0016ETP), Module 2 (GL20-1600END)
//     wf2_do [GL20-RTU-ECT_1.3.5.0]
//       modules: Module 1 (GL20-0016ETP), Module 2 (GL20-1600END)
//     wf1_do [GL20-RTU-ECT_1.3.5.0]
//       modules: Module 1 (GL20-0016ETP), Module 2 (GL20-1600END)
//     wf0_do [GL20-RTU-ECT_1.3.5.0]
//       modules: Module 1 (GL20-0016ETP), Module 2 (GL20-1600END)
//   DEVICE pm side, AmsNetId 192.168.11.159.5.1
//     Box 49 (CU2508) [CU2508 Ethernet Port]
//     lb0_dio [GL20-RTU-ECT_1.3.5.0]
//       modules: Module 1 (GL20-1600END), Module 2 (GL20-0016ETP)
//     lb0_converter [MD800_ECAT_9Axis_V0.19]
//     lc0_dio [GL20-RTU-ECT_1.3.5.0]
//       modules: Module 1 (GL20-1600END), Module 2 (GL20-1600END), Module 3 (GL20-0016ETP), Module 4 (GL20-0016ETP)
//     lc0_converter [MD800_ECAT_9Axis_V0.19]
//     lc0_servermoter [SV630_1Axis_03713]
//     pm0_1_dio [GL20-RTU-ECT_1.3.5.0]
//       modules: Module 1 (GL20-1600END), Module 2 (GL20-1600END), Module 3 (GL20-1600END), Module 4 (GL20-1600END), Module 5 (GL20-1600END), Module 6 (GL20-0016ETP), Module 7 (GL20-0016ETP)
//     pm0_1_innerConv [MD800_ECAT_9Axis_V0.19]
//     pm0_1_outerConv [MD800_ECAT_9Axis_V0.19]
//     pm0_buf0 [SV630_1Axis_03713]
//     pm0_buf1 [SV630_1Axis_03713]
//     pm1_buf0 [SV630_1Axis_03713]
//     pm1_buf1 [SV630_1Axis_03713]
//     pm0_1_RFID [SIG350-0006AP100]
//       modules: Module 1 (IOL_32/32_I/O-Bytes), Module 2 (IOL_32/32_I/O-Bytes), Module 3 (IOL_32/32_I/O-Bytes), Module 4 (IOL_32/32_I/O-Bytes), Module 5 (Slot Empty), Module 6 (Slot Empty), Module 7 (Slot Empty), Module 8 (Slot Empty)
//     fr0_dio [GL20-RTU-ECT_1.3.5.0]
//       modules: Module 1 (GL20-1600END), Module 2 (GL20-0016ETP)
//     fr0_servermotor [SV630_1Axis_03713]
//     pm2_3_dio [GL20-RTU-ECT_1.3.5.0]
//       modules: Module 1 (GL20-1600END), Module 2 (GL20-1600END), Module 3 (GL20-1600END), Module 4 (GL20-1600END), Module 5 (GL20-1600END), Module 6 (GL20-1600END), Module 7 (GL20-0016ETP), Module 8 (GL20-0016ETP)
//     pm2_3_innerConv [MD800_ECAT_9Axis_V0.19]
//     pm2_3_outerConv [MD800_ECAT_9Axis_V0.19]
//     pm2_buf0 [SV630_1Axis_03713]
//     pm2_buf1 [SV630_1Axis_03713]
//     pm3_buf0 [SV630_1Axis_03713]
//     pm3_buf1 [SV630_1Axis_03713]
//     pm2_3_RFID [SIG350-0006AP100]
//       modules: Module 1 (IOL_32/32_I/O-Bytes), Module 2 (IOL_32/32_I/O-Bytes), Module 3 (IOL_32/32_I/O-Bytes), Module 4 (IOL_32/32_I/O-Bytes), Module 5 (Slot Empty), Module 6 (Slot Empty), Module 7 (Slot Empty), Module 8 (Slot Empty)
//     pm4_5_dio [GL20-RTU-ECT_1.3.5.0]
//       modules: Module 1 (GL20-1600END), Module 2 (GL20-1600END), Module 3 (GL20-1600END), Module 4 (GL20-1600END), Module 5 (GL20-1600END), Module 6 (GL20-1600END), Module 7 (GL20-0016ETP), Module 8 (GL20-0016ETP)
//     pm4_5_innerConv [MD800_ECAT_9Axis_V0.19]
//     pm4_5_outerConv [MD800_ECAT_9Axis_V0.19]
//     pm4_buf0 [SV630_1Axis_03713]
//     pm4_buf1 [SV630_1Axis_03713]
//     pm5_buf0 [SV630_1Axis_03713]
//     pm5_buf1 [SV630_1Axis_03713]
//     pm4_5_RFID [SIG350-0006AP100]
//       modules: Module 1 (IOL_32/32_I/O-Bytes), Module 2 (IOL_32/32_I/O-Bytes), Module 3 (IOL_32/32_I/O-Bytes), Module 4 (IOL_32/32_I/O-Bytes), Module 5 (Slot Empty), Module 6 (Slot Empty), Module 7 (Slot Empty), Module 8 (Slot Empty)
//     pm6_7_dio [GL20-RTU-ECT_1.3.5.0]
//       modules: Module 1 (GL20-1600END), Module 2 (GL20-1600END), Module 3 (GL20-1600END), Module 4 (GL20-1600END), Module 5 (GL20-1600END), Module 6 (GL20-0016ETP), Module 7 (GL20-0016ETP)
//     pm6_7_innerConv [MD800_ECAT_9Axis_V0.19]
//     pm6_7_outerConv [MD800_ECAT_9Axis_V0.19]
//     pm6_buf0 [SV630_1Axis_03713]
//     pm6_buf1 [SV630_1Axis_03713]
//     pm7_buf0 [SV630_1Axis_03713]
//     pm7_buf1 [SV630_1Axis_03713]
//     pm6_7_RFID [SIG350-0006AP100]
//       modules: Module 1 (IOL_32/32_I/O-Bytes), Module 2 (IOL_32/32_I/O-Bytes), Module 3 (IOL_32/32_I/O-Bytes), Module 4 (IOL_32/32_I/O-Bytes), Module 5 (Slot Empty), Module 6 (Slot Empty), Module 7 (Slot Empty), Module 8 (Slot Empty)
//     fr1_dio [GL20-RTU-ECT_1.3.5.0]
//       modules: Module 1 (GL20-1600END), Module 2 (GL20-0016ETP)
//     fr1_servermotor [SV630_1Axis_03713]
//     pm8_9_dio [GL20-RTU-ECT_1.3.5.0]
//       modules: Module 1 (GL20-1600END), Module 2 (GL20-1600END), Module 3 (GL20-1600END), Module 4 (GL20-1600END), Module 5 (GL20-1600END), Module 6 (GL20-0016ETP), Module 7 (GL20-0016ETP)
//     pm8_9_innerConv [MD800_ECAT_9Axis_V0.19]
//     pm8_9_outerConv [MD800_ECAT_9Axis_V0.19]
//     pm8_buf0 [SV630_1Axis_03713]
//     pm8_buf1 [SV630_1Axis_03713]
//     pm9_buf0 [SV630_1Axis_03713]
//     pm9_buf1 [SV630_1Axis_03713]
//     pm8_9_RFID [SIG350-0006AP100]
//       modules: Module 1 (IOL_32/32_I/O-Bytes), Module 2 (IOL_32/32_I/O-Bytes), Module 3 (IOL_32/32_I/O-Bytes), Module 4 (IOL_32/32_I/O-Bytes), Module 5 (Slot Empty), Module 6 (Slot Empty), Module 7 (Slot Empty), Module 8 (Slot Empty)
//     lb1_dio [GL20-RTU-ECT_1.3.5.0]
//       modules: Module 1 (GL20-1600END), Module 2 (GL20-0016ETP)
//     lb1_converter [MD800_ECAT_9Axis_V0.19]
//     lc1_dio [GL20-RTU-ECT_1.3.5.0]
//       modules: Module 1 (GL20-1600END), Module 2 (GL20-1600END), Module 3 (GL20-0016ETP), Module 4 (GL20-0016ETP)
//     lc1_converter [MD800_ECAT_9Axis_V0.19]
//     lc1_servermoter [SV630_1Axis_03713]
//   DEVICE Device 5 (USB)
//     Box 1 (CX2100 Power Supply)
//   DEVICE Device 6 (COM Port)
//   DEVICE Device 7 (NOV-DP-RAM)
//   DEVICE Device 8 (EtherCAT) (disabled), AmsNetId 192.168.11.159.9.1
//     Box 63 (DL-EC1A) [DL-EC1A]
// variable links:
//   NC-Task 1 SAF/Axes/fr0 <-> pm side/fr0_servermotor
//     Drive/Inputs/In/nDataIn1 <-> Inputs/Following error actual value
//     Drive/Inputs/In/nDataIn3[0] <-> Inputs/Torque actual value
//     Drive/Inputs/In/nDcOutputTime <-> InfoData/DcOutputShift
//     Drive/Inputs/In/nState1 <-> Inputs/Statusword
//     Drive/Inputs/In/nState2 <-> Inputs/Statusword @bit 8
//     Drive/Inputs/In/nState4 @bit 1 <-> WcState/InputToggle
//     Drive/Inputs/In/nState4 <-> WcState/WcState
//     Drive/Outputs/Out/nCtrl1 <-> Outputs/Controlword
//     Drive/Outputs/Out/nCtrl2 <-> Outputs/Controlword @bit 8
//     Drive/Outputs/Out/nDataOut1 <-> Outputs/Target position
//     Enc/Inputs/In/nDataIn1 <-> Inputs/Position actual value
//     Enc/Inputs/In/nDataIn3 <-> Inputs/Touch probe pos1 pos value
//     Enc/Inputs/In/nDataIn5 <-> Inputs/Touch probe pos2 pos value
//     Enc/Inputs/In/nDcInputTime <-> InfoData/DcInputShift
//     Enc/Inputs/In/nState4 @bit 1 <-> WcState/InputToggle
//     Enc/Inputs/In/nState4 <-> WcState/WcState
//     Enc/Inputs/In/nState5 <-> Inputs/Touch probe status
//     Enc/Inputs/In/nState6 <-> Inputs/Touch probe status @bit 8
//     Enc/Outputs/Out/nCtrl5 <-> Outputs/Touch probe function
//     Enc/Outputs/Out/nCtrl6 <-> Outputs/Touch probe function @bit 8
//   NC-Task 1 SAF/Axes/fr1 <-> pm side/fr1_servermotor
//     Drive/Inputs/In/nDataIn1 <-> Inputs/Following error actual value
//     Drive/Inputs/In/nDataIn3[0] <-> Inputs/Torque actual value
//     Drive/Inputs/In/nDcOutputTime <-> InfoData/DcOutputShift
//     Drive/Inputs/In/nState1 <-> Inputs/Statusword
//     Drive/Inputs/In/nState2 <-> Inputs/Statusword @bit 8
//     Drive/Inputs/In/nState4 @bit 1 <-> WcState/InputToggle
//     Drive/Inputs/In/nState4 <-> WcState/WcState
//     Drive/Outputs/Out/nCtrl1 <-> Outputs/Controlword
//     Drive/Outputs/Out/nCtrl2 <-> Outputs/Controlword @bit 8
//     Drive/Outputs/Out/nDataOut1 <-> Outputs/Target position
//     Enc/Inputs/In/nDataIn1 <-> Inputs/Position actual value
//     Enc/Inputs/In/nDataIn3 <-> Inputs/Touch probe pos1 pos value
//     Enc/Inputs/In/nDataIn5 <-> Inputs/Touch probe pos2 pos value
//     Enc/Inputs/In/nDcInputTime <-> InfoData/DcInputShift
//     Enc/Inputs/In/nState4 @bit 1 <-> WcState/InputToggle
//     Enc/Inputs/In/nState4 <-> WcState/WcState
//     Enc/Inputs/In/nState5 <-> Inputs/Touch probe status
//     Enc/Inputs/In/nState6 <-> Inputs/Touch probe status @bit 8
//     Enc/Outputs/Out/nCtrl5 <-> Outputs/Touch probe function
//     Enc/Outputs/Out/nCtrl6 <-> Outputs/Touch probe function @bit 8
//   NC-Task 1 SAF/Axes/lc0 <-> pm side/lc0_servermoter
//     Drive/Inputs/In/nDataIn1 <-> Inputs/Following error actual value
//     Drive/Inputs/In/nDataIn3[0] <-> Inputs/Torque actual value
//     Drive/Inputs/In/nDcOutputTime <-> InfoData/DcOutputShift
//     Drive/Inputs/In/nState1 <-> Inputs/Statusword
//     Drive/Inputs/In/nState2 <-> Inputs/Statusword @bit 8
//     Drive/Inputs/In/nState4 @bit 1 <-> WcState/InputToggle
//     Drive/Inputs/In/nState4 <-> WcState/WcState
//     Drive/Outputs/Out/nCtrl1 <-> Outputs/Controlword
//     Drive/Outputs/Out/nCtrl2 <-> Outputs/Controlword @bit 8
//     Drive/Outputs/Out/nDataOut1 <-> Outputs/Target position
//     Enc/Inputs/In/nDataIn1 <-> Inputs/Position actual value
//     Enc/Inputs/In/nDataIn3 <-> Inputs/Touch probe pos1 pos value
//     Enc/Inputs/In/nDataIn5 <-> Inputs/Touch probe pos2 pos value
//     Enc/Inputs/In/nDcInputTime <-> InfoData/DcInputShift
//     Enc/Inputs/In/nState4 @bit 1 <-> WcState/InputToggle
//     Enc/Inputs/In/nState4 <-> WcState/WcState
//     Enc/Inputs/In/nState5 <-> Inputs/Touch probe status
//     Enc/Inputs/In/nState6 <-> Inputs/Touch probe status @bit 8
//     Enc/Outputs/Out/nCtrl5 <-> Outputs/Touch probe function
//     Enc/Outputs/Out/nCtrl6 <-> Outputs/Touch probe function @bit 8
//   NC-Task 1 SAF/Axes/lc1 <-> pm side/lc1_servermoter
//     Drive/Inputs/In/nDataIn1 <-> Inputs/Following error actual value
//     Drive/Inputs/In/nDataIn3[0] <-> Inputs/Torque actual value
//     Drive/Inputs/In/nDcOutputTime <-> InfoData/DcOutputShift
//     Drive/Inputs/In/nState1 <-> Inputs/Statusword
//     Drive/Inputs/In/nState2 <-> Inputs/Statusword @bit 8
//     Drive/Inputs/In/nState4 @bit 1 <-> WcState/InputToggle
//     Drive/Inputs/In/nState4 <-> WcState/WcState
//     Drive/Outputs/Out/nCtrl1 <-> Outputs/Controlword
//     Drive/Outputs/Out/nCtrl2 <-> Outputs/Controlword @bit 8
//     Drive/Outputs/Out/nDataOut1 <-> Outputs/Target position
//     Enc/Inputs/In/nDataIn1 <-> Inputs/Position actual value
//     Enc/Inputs/In/nDataIn3 <-> Inputs/Touch probe pos1 pos value
//     Enc/Inputs/In/nDataIn5 <-> Inputs/Touch probe pos2 pos value
//     Enc/Inputs/In/nDcInputTime <-> InfoData/DcInputShift
//     Enc/Inputs/In/nState4 @bit 1 <-> WcState/InputToggle
//     Enc/Inputs/In/nState4 <-> WcState/WcState
//     Enc/Inputs/In/nState5 <-> Inputs/Touch probe status
//     Enc/Inputs/In/nState6 <-> Inputs/Touch probe status @bit 8
//     Enc/Outputs/Out/nCtrl5 <-> Outputs/Touch probe function
//     Enc/Outputs/Out/nCtrl6 <-> Outputs/Touch probe function @bit 8
//   NC-Task 1 SAF/Axes/pm0_buf0 <-> pm side/pm0_buf0
//     Drive/Inputs/In/nDataIn1 <-> Inputs/Following error actual value
//     Drive/Inputs/In/nDataIn3[0] <-> Inputs/Torque actual value
//     Drive/Inputs/In/nDcOutputTime <-> InfoData/DcOutputShift
//     Drive/Inputs/In/nState1 <-> Inputs/Statusword
//     Drive/Inputs/In/nState2 <-> Inputs/Statusword @bit 8
//     Drive/Inputs/In/nState4 @bit 1 <-> WcState/InputToggle
//     Drive/Inputs/In/nState4 <-> WcState/WcState
//     Drive/Outputs/Out/nCtrl1 <-> Outputs/Controlword
//     Drive/Outputs/Out/nCtrl2 <-> Outputs/Controlword @bit 8
//     Drive/Outputs/Out/nDataOut1 <-> Outputs/Target position
//     Enc/Inputs/In/nDataIn1 <-> Inputs/Position actual value
//     Enc/Inputs/In/nDataIn3 <-> Inputs/Touch probe pos1 pos value
//     Enc/Inputs/In/nDataIn5 <-> Inputs/Touch probe pos2 pos value
//     Enc/Inputs/In/nDcInputTime <-> InfoData/DcInputShift
//     Enc/Inputs/In/nState4 @bit 1 <-> WcState/InputToggle
//     Enc/Inputs/In/nState4 <-> WcState/WcState
//     Enc/Inputs/In/nState5 <-> Inputs/Touch probe status
//     Enc/Inputs/In/nState6 <-> Inputs/Touch probe status @bit 8
//     Enc/Outputs/Out/nCtrl5 <-> Outputs/Touch probe function
//     Enc/Outputs/Out/nCtrl6 <-> Outputs/Touch probe function @bit 8
//   NC-Task 1 SAF/Axes/pm0_buf1 <-> pm side/pm0_buf1
//     Drive/Inputs/In/nDataIn1 <-> Inputs/Following error actual value
//     Drive/Inputs/In/nDataIn3[0] <-> Inputs/Torque actual value
//     Drive/Inputs/In/nDcOutputTime <-> InfoData/DcOutputShift
//     Drive/Inputs/In/nState1 <-> Inputs/Statusword
//     Drive/Inputs/In/nState2 <-> Inputs/Statusword @bit 8
//     Drive/Inputs/In/nState4 @bit 1 <-> WcState/InputToggle
//     Drive/Inputs/In/nState4 <-> WcState/WcState
//     Drive/Outputs/Out/nCtrl1 <-> Outputs/Controlword
//     Drive/Outputs/Out/nCtrl2 <-> Outputs/Controlword @bit 8
//     Drive/Outputs/Out/nDataOut1 <-> Outputs/Target position
//     Enc/Inputs/In/nDataIn1 <-> Inputs/Position actual value
//     Enc/Inputs/In/nDataIn3 <-> Inputs/Touch probe pos1 pos value
//     Enc/Inputs/In/nDataIn5 <-> Inputs/Touch probe pos2 pos value
//     Enc/Inputs/In/nDcInputTime <-> InfoData/DcInputShift
//     Enc/Inputs/In/nState4 @bit 1 <-> WcState/InputToggle
//     Enc/Inputs/In/nState4 <-> WcState/WcState
//     Enc/Inputs/In/nState5 <-> Inputs/Touch probe status
//     Enc/Inputs/In/nState6 <-> Inputs/Touch probe status @bit 8
//     Enc/Outputs/Out/nCtrl5 <-> Outputs/Touch probe function
//     Enc/Outputs/Out/nCtrl6 <-> Outputs/Touch probe function @bit 8
//   NC-Task 1 SAF/Axes/pm1_buf0 <-> pm side/pm1_buf0
//     Drive/Inputs/In/nDataIn1 <-> Inputs/Following error actual value
//     Drive/Inputs/In/nDataIn3[0] <-> Inputs/Torque actual value
//     Drive/Inputs/In/nDcOutputTime <-> InfoData/DcOutputShift
//     Drive/Inputs/In/nState1 <-> Inputs/Statusword
//     Drive/Inputs/In/nState2 <-> Inputs/Statusword @bit 8
//     Drive/Inputs/In/nState4 @bit 1 <-> WcState/InputToggle
//     Drive/Inputs/In/nState4 <-> WcState/WcState
//     Drive/Outputs/Out/nCtrl1 <-> Outputs/Controlword
//     Drive/Outputs/Out/nCtrl2 <-> Outputs/Controlword @bit 8
//     Drive/Outputs/Out/nDataOut1 <-> Outputs/Target position
//     Enc/Inputs/In/nDataIn1 <-> Inputs/Position actual value
//     Enc/Inputs/In/nDataIn3 <-> Inputs/Touch probe pos1 pos value
//     Enc/Inputs/In/nDataIn5 <-> Inputs/Touch probe pos2 pos value
//     Enc/Inputs/In/nDcInputTime <-> InfoData/DcInputShift
//     Enc/Inputs/In/nState4 @bit 1 <-> WcState/InputToggle
//     Enc/Inputs/In/nState4 <-> WcState/WcState
//     Enc/Inputs/In/nState5 <-> Inputs/Touch probe status
//     Enc/Inputs/In/nState6 <-> Inputs/Touch probe status @bit 8
//     Enc/Outputs/Out/nCtrl5 <-> Outputs/Touch probe function
//     Enc/Outputs/Out/nCtrl6 <-> Outputs/Touch probe function @bit 8
//   NC-Task 1 SAF/Axes/pm1_buf1 <-> pm side/pm1_buf1
//     Drive/Inputs/In/nDataIn1 <-> Inputs/Following error actual value
//     Drive/Inputs/In/nDataIn3[0] <-> Inputs/Torque actual value
//     Drive/Inputs/In/nDcOutputTime <-> InfoData/DcOutputShift
//     Drive/Inputs/In/nState1 <-> Inputs/Statusword
//     Drive/Inputs/In/nState2 <-> Inputs/Statusword @bit 8
//     Drive/Inputs/In/nState4 @bit 1 <-> WcState/InputToggle
//     Drive/Inputs/In/nState4 <-> WcState/WcState
//     Drive/Outputs/Out/nCtrl1 <-> Outputs/Controlword
//     Drive/Outputs/Out/nCtrl2 <-> Outputs/Controlword @bit 8
//     Drive/Outputs/Out/nDataOut1 <-> Outputs/Target position
//     Enc/Inputs/In/nDataIn1 <-> Inputs/Position actual value
//     Enc/Inputs/In/nDataIn3 <-> Inputs/Touch probe pos1 pos value
//     Enc/Inputs/In/nDataIn5 <-> Inputs/Touch probe pos2 pos value
//     Enc/Inputs/In/nDcInputTime <-> InfoData/DcInputShift
//     Enc/Inputs/In/nState4 @bit 1 <-> WcState/InputToggle
//     Enc/Inputs/In/nState4 <-> WcState/WcState
//     Enc/Inputs/In/nState5 <-> Inputs/Touch probe status
//     Enc/Inputs/In/nState6 <-> Inputs/Touch probe status @bit 8
//     Enc/Outputs/Out/nCtrl5 <-> Outputs/Touch probe function
//     Enc/Outputs/Out/nCtrl6 <-> Outputs/Touch probe function @bit 8
//   NC-Task 1 SAF/Axes/pm2_buf0 <-> pm side/pm2_buf0
//     Drive/Inputs/In/nDataIn1 <-> Inputs/Following error actual value
//     Drive/Inputs/In/nDataIn3[0] <-> Inputs/Torque actual value
//     Drive/Inputs/In/nDcOutputTime <-> InfoData/DcOutputShift
//     Drive/Inputs/In/nState1 <-> Inputs/Statusword
//     Drive/Inputs/In/nState2 <-> Inputs/Statusword @bit 8
//     Drive/Inputs/In/nState4 @bit 1 <-> WcState/InputToggle
//     Drive/Inputs/In/nState4 <-> WcState/WcState
//     Drive/Outputs/Out/nCtrl1 <-> Outputs/Controlword
//     Drive/Outputs/Out/nCtrl2 <-> Outputs/Controlword @bit 8
//     Drive/Outputs/Out/nDataOut1 <-> Outputs/Target position
//     Enc/Inputs/In/nDataIn1 <-> Inputs/Position actual value
//     Enc/Inputs/In/nDataIn3 <-> Inputs/Touch probe pos1 pos value
//     Enc/Inputs/In/nDataIn5 <-> Inputs/Touch probe pos2 pos value
//     Enc/Inputs/In/nDcInputTime <-> InfoData/DcInputShift
//     Enc/Inputs/In/nState4 @bit 1 <-> WcState/InputToggle
//     Enc/Inputs/In/nState4 <-> WcState/WcState
//     Enc/Inputs/In/nState5 <-> Inputs/Touch probe status
//     Enc/Inputs/In/nState6 <-> Inputs/Touch probe status @bit 8
//     Enc/Outputs/Out/nCtrl5 <-> Outputs/Touch probe function
//     Enc/Outputs/Out/nCtrl6 <-> Outputs/Touch probe function @bit 8
//   NC-Task 1 SAF/Axes/pm2_buf1 <-> pm side/pm2_buf1
//     Drive/Inputs/In/nDataIn1 <-> Inputs/Following error actual value
//     Drive/Inputs/In/nDataIn3[0] <-> Inputs/Torque actual value
//     Drive/Inputs/In/nDcOutputTime <-> InfoData/DcOutputShift
//     Drive/Inputs/In/nState1 <-> Inputs/Statusword
//     Drive/Inputs/In/nState2 <-> Inputs/Statusword @bit 8
//     Drive/Inputs/In/nState4 @bit 1 <-> WcState/InputToggle
//     Drive/Inputs/In/nState4 <-> WcState/WcState
//     Drive/Outputs/Out/nCtrl1 <-> Outputs/Controlword
//     Drive/Outputs/Out/nCtrl2 <-> Outputs/Controlword @bit 8
//     Drive/Outputs/Out/nDataOut1 <-> Outputs/Target position
//     Enc/Inputs/In/nDataIn1 <-> Inputs/Position actual value
//     Enc/Inputs/In/nDataIn3 <-> Inputs/Touch probe pos1 pos value
//     Enc/Inputs/In/nDataIn5 <-> Inputs/Touch probe pos2 pos value
//     Enc/Inputs/In/nDcInputTime <-> InfoData/DcInputShift
//     Enc/Inputs/In/nState4 @bit 1 <-> WcState/InputToggle
//     Enc/Inputs/In/nState4 <-> WcState/WcState
//     Enc/Inputs/In/nState5 <-> Inputs/Touch probe status
//     Enc/Inputs/In/nState6 <-> Inputs/Touch probe status @bit 8
//     Enc/Outputs/Out/nCtrl5 <-> Outputs/Touch probe function
//     Enc/Outputs/Out/nCtrl6 <-> Outputs/Touch probe function @bit 8
//   NC-Task 1 SAF/Axes/pm3_buf0 <-> pm side/pm3_buf0
//     Drive/Inputs/In/nDataIn1 <-> Inputs/Following error actual value
//     Drive/Inputs/In/nDataIn3[0] <-> Inputs/Torque actual value
//     Drive/Inputs/In/nDcOutputTime <-> InfoData/DcOutputShift
//     Drive/Inputs/In/nState1 <-> Inputs/Statusword
//     Drive/Inputs/In/nState2 <-> Inputs/Statusword @bit 8
//     Drive/Inputs/In/nState4 @bit 1 <-> WcState/InputToggle
//     Drive/Inputs/In/nState4 <-> WcState/WcState
//     Drive/Outputs/Out/nCtrl1 <-> Outputs/Controlword
//     Drive/Outputs/Out/nCtrl2 <-> Outputs/Controlword @bit 8
//     Drive/Outputs/Out/nDataOut1 <-> Outputs/Target position
//     Enc/Inputs/In/nDataIn1 <-> Inputs/Position actual value
//     Enc/Inputs/In/nDataIn3 <-> Inputs/Touch probe pos1 pos value
//     Enc/Inputs/In/nDataIn5 <-> Inputs/Touch probe pos2 pos value
//     Enc/Inputs/In/nDcInputTime <-> InfoData/DcInputShift
//     Enc/Inputs/In/nState4 @bit 1 <-> WcState/InputToggle
//     Enc/Inputs/In/nState4 <-> WcState/WcState
//     Enc/Inputs/In/nState5 <-> Inputs/Touch probe status
//     Enc/Inputs/In/nState6 <-> Inputs/Touch probe status @bit 8
//     Enc/Outputs/Out/nCtrl5 <-> Outputs/Touch probe function
//     Enc/Outputs/Out/nCtrl6 <-> Outputs/Touch probe function @bit 8
//   NC-Task 1 SAF/Axes/pm3_buf1 <-> pm side/pm3_buf1
//     Drive/Inputs/In/nDataIn1 <-> Inputs/Following error actual value
//     Drive/Inputs/In/nDataIn3[0] <-> Inputs/Torque actual value
//     Drive/Inputs/In/nDcOutputTime <-> InfoData/DcOutputShift
//     Drive/Inputs/In/nState1 <-> Inputs/Statusword
//     Drive/Inputs/In/nState2 <-> Inputs/Statusword @bit 8
//     Drive/Inputs/In/nState4 @bit 1 <-> WcState/InputToggle
//     Drive/Inputs/In/nState4 <-> WcState/WcState
//     Drive/Outputs/Out/nCtrl1 <-> Outputs/Controlword
//     Drive/Outputs/Out/nCtrl2 <-> Outputs/Controlword @bit 8
//     Drive/Outputs/Out/nDataOut1 <-> Outputs/Target position
//     Enc/Inputs/In/nDataIn1 <-> Inputs/Position actual value
//     Enc/Inputs/In/nDataIn3 <-> Inputs/Touch probe pos1 pos value
//     Enc/Inputs/In/nDataIn5 <-> Inputs/Touch probe pos2 pos value
//     Enc/Inputs/In/nDcInputTime <-> InfoData/DcInputShift
//     Enc/Inputs/In/nState4 @bit 1 <-> WcState/InputToggle
//     Enc/Inputs/In/nState4 <-> WcState/WcState
//     Enc/Inputs/In/nState5 <-> Inputs/Touch probe status
//     Enc/Inputs/In/nState6 <-> Inputs/Touch probe status @bit 8
//     Enc/Outputs/Out/nCtrl5 <-> Outputs/Touch probe function
//     Enc/Outputs/Out/nCtrl6 <-> Outputs/Touch probe function @bit 8
//   NC-Task 1 SAF/Axes/pm4_buf0 <-> pm side/pm4_buf0
//     Drive/Inputs/In/nDataIn1 <-> Inputs/Following error actual value
//     Drive/Inputs/In/nDataIn3[0] <-> Inputs/Torque actual value
//     Drive/Inputs/In/nDcOutputTime <-> InfoData/DcOutputShift
//     Drive/Inputs/In/nState1 <-> Inputs/Statusword
//     Drive/Inputs/In/nState2 <-> Inputs/Statusword @bit 8
//     Drive/Inputs/In/nState4 @bit 1 <-> WcState/InputToggle
//     Drive/Inputs/In/nState4 <-> WcState/WcState
//     Drive/Outputs/Out/nCtrl1 <-> Outputs/Controlword
//     Drive/Outputs/Out/nCtrl2 <-> Outputs/Controlword @bit 8
//     Drive/Outputs/Out/nDataOut1 <-> Outputs/Target position
//     Enc/Inputs/In/nDataIn1 <-> Inputs/Position actual value
//     Enc/Inputs/In/nDataIn3 <-> Inputs/Touch probe pos1 pos value
//     Enc/Inputs/In/nDataIn5 <-> Inputs/Touch probe pos2 pos value
//     Enc/Inputs/In/nDcInputTime <-> InfoData/DcInputShift
//     Enc/Inputs/In/nState4 @bit 1 <-> WcState/InputToggle
//     Enc/Inputs/In/nState4 <-> WcState/WcState
//     Enc/Inputs/In/nState5 <-> Inputs/Touch probe status
//     Enc/Inputs/In/nState6 <-> Inputs/Touch probe status @bit 8
//     Enc/Outputs/Out/nCtrl5 <-> Outputs/Touch probe function
//     Enc/Outputs/Out/nCtrl6 <-> Outputs/Touch probe function @bit 8
//   NC-Task 1 SAF/Axes/pm4_buf1 <-> pm side/pm4_buf1
//     Drive/Inputs/In/nDataIn1 <-> Inputs/Following error actual value
//     Drive/Inputs/In/nDataIn3[0] <-> Inputs/Torque actual value
//     Drive/Inputs/In/nDcOutputTime <-> InfoData/DcOutputShift
//     Drive/Inputs/In/nState1 <-> Inputs/Statusword
//     Drive/Inputs/In/nState2 <-> Inputs/Statusword @bit 8
//     Drive/Inputs/In/nState4 @bit 1 <-> WcState/InputToggle
//     Drive/Inputs/In/nState4 <-> WcState/WcState
//     Drive/Outputs/Out/nCtrl1 <-> Outputs/Controlword
//     Drive/Outputs/Out/nCtrl2 <-> Outputs/Controlword @bit 8
//     Drive/Outputs/Out/nDataOut1 <-> Outputs/Target position
//     Enc/Inputs/In/nDataIn1 <-> Inputs/Position actual value
//     Enc/Inputs/In/nDataIn3 <-> Inputs/Touch probe pos1 pos value
//     Enc/Inputs/In/nDataIn5 <-> Inputs/Touch probe pos2 pos value
//     Enc/Inputs/In/nDcInputTime <-> InfoData/DcInputShift
//     Enc/Inputs/In/nState4 @bit 1 <-> WcState/InputToggle
//     Enc/Inputs/In/nState4 <-> WcState/WcState
//     Enc/Inputs/In/nState5 <-> Inputs/Touch probe status
//     Enc/Inputs/In/nState6 <-> Inputs/Touch probe status @bit 8
//     Enc/Outputs/Out/nCtrl5 <-> Outputs/Touch probe function
//     Enc/Outputs/Out/nCtrl6 <-> Outputs/Touch probe function @bit 8
//   NC-Task 1 SAF/Axes/pm5_buf0 <-> pm side/pm5_buf0
//     Drive/Inputs/In/nDataIn1 <-> Inputs/Following error actual value
//     Drive/Inputs/In/nDataIn3[0] <-> Inputs/Torque actual value
//     Drive/Inputs/In/nDcOutputTime <-> InfoData/DcOutputShift
//     Drive/Inputs/In/nState1 <-> Inputs/Statusword
//     Drive/Inputs/In/nState2 <-> Inputs/Statusword @bit 8
//     Drive/Inputs/In/nState4 @bit 1 <-> WcState/InputToggle
//     Drive/Inputs/In/nState4 <-> WcState/WcState
//     Drive/Outputs/Out/nCtrl1 <-> Outputs/Controlword
//     Drive/Outputs/Out/nCtrl2 <-> Outputs/Controlword @bit 8
//     Drive/Outputs/Out/nDataOut1 <-> Outputs/Target position
//     Enc/Inputs/In/nDataIn1 <-> Inputs/Position actual value
//     Enc/Inputs/In/nDataIn3 <-> Inputs/Touch probe pos1 pos value
//     Enc/Inputs/In/nDataIn5 <-> Inputs/Touch probe pos2 pos value
//     Enc/Inputs/In/nDcInputTime <-> InfoData/DcInputShift
//     Enc/Inputs/In/nState4 @bit 1 <-> WcState/InputToggle
//     Enc/Inputs/In/nState4 <-> WcState/WcState
//     Enc/Inputs/In/nState5 <-> Inputs/Touch probe status
//     Enc/Inputs/In/nState6 <-> Inputs/Touch probe status @bit 8
//     Enc/Outputs/Out/nCtrl5 <-> Outputs/Touch probe function
//     Enc/Outputs/Out/nCtrl6 <-> Outputs/Touch probe function @bit 8
//   NC-Task 1 SAF/Axes/pm5_buf1 <-> pm side/pm5_buf1
//     Drive/Inputs/In/nDataIn1 <-> Inputs/Following error actual value
//     Drive/Inputs/In/nDataIn3[0] <-> Inputs/Torque actual value
//     Drive/Inputs/In/nDcOutputTime <-> InfoData/DcOutputShift
//     Drive/Inputs/In/nState1 <-> Inputs/Statusword
//     Drive/Inputs/In/nState2 <-> Inputs/Statusword @bit 8
//     Drive/Inputs/In/nState4 @bit 1 <-> WcState/InputToggle
//     Drive/Inputs/In/nState4 <-> WcState/WcState
//     Drive/Outputs/Out/nCtrl1 <-> Outputs/Controlword
//     Drive/Outputs/Out/nCtrl2 <-> Outputs/Controlword @bit 8
//     Drive/Outputs/Out/nDataOut1 <-> Outputs/Target position
//     Enc/Inputs/In/nDataIn1 <-> Inputs/Position actual value
//     Enc/Inputs/In/nDataIn3 <-> Inputs/Touch probe pos1 pos value
//     Enc/Inputs/In/nDataIn5 <-> Inputs/Touch probe pos2 pos value
//     Enc/Inputs/In/nDcInputTime <-> InfoData/DcInputShift
//     Enc/Inputs/In/nState4 @bit 1 <-> WcState/InputToggle
//     Enc/Inputs/In/nState4 <-> WcState/WcState
//     Enc/Inputs/In/nState5 <-> Inputs/Touch probe status
//     Enc/Inputs/In/nState6 <-> Inputs/Touch probe status @bit 8
//     Enc/Outputs/Out/nCtrl5 <-> Outputs/Touch probe function
//     Enc/Outputs/Out/nCtrl6 <-> Outputs/Touch probe function @bit 8
//   NC-Task 1 SAF/Axes/pm6_buf0 <-> pm side/pm6_buf0
//     Drive/Inputs/In/nDataIn1 <-> Inputs/Following error actual value
//     Drive/Inputs/In/nDataIn3[0] <-> Inputs/Torque actual value
//     Drive/Inputs/In/nDcOutputTime <-> InfoData/DcOutputShift
//     Drive/Inputs/In/nState1 <-> Inputs/Statusword
//     Drive/Inputs/In/nState2 <-> Inputs/Statusword @bit 8
//     Drive/Inputs/In/nState4 @bit 1 <-> WcState/InputToggle
//     Drive/Inputs/In/nState4 <-> WcState/WcState
//     Drive/Outputs/Out/nCtrl1 <-> Outputs/Controlword
//     Drive/Outputs/Out/nCtrl2 <-> Outputs/Controlword @bit 8
//     Drive/Outputs/Out/nDataOut1 <-> Outputs/Target position
//     Enc/Inputs/In/nDataIn1 <-> Inputs/Position actual value
//     Enc/Inputs/In/nDataIn3 <-> Inputs/Touch probe pos1 pos value
//     Enc/Inputs/In/nDataIn5 <-> Inputs/Touch probe pos2 pos value
//     Enc/Inputs/In/nDcInputTime <-> InfoData/DcInputShift
//     Enc/Inputs/In/nState4 @bit 1 <-> WcState/InputToggle
//     Enc/Inputs/In/nState4 <-> WcState/WcState
//     Enc/Inputs/In/nState5 <-> Inputs/Touch probe status
//     Enc/Inputs/In/nState6 <-> Inputs/Touch probe status @bit 8
//     Enc/Outputs/Out/nCtrl5 <-> Outputs/Touch probe function
//     Enc/Outputs/Out/nCtrl6 <-> Outputs/Touch probe function @bit 8
//   NC-Task 1 SAF/Axes/pm6_buf1 <-> pm side/pm6_buf1
//     Drive/Inputs/In/nDataIn1 <-> Inputs/Following error actual value
//     Drive/Inputs/In/nDataIn3[0] <-> Inputs/Torque actual value
//     Drive/Inputs/In/nDcOutputTime <-> InfoData/DcOutputShift
//     Drive/Inputs/In/nState1 <-> Inputs/Statusword
//     Drive/Inputs/In/nState2 <-> Inputs/Statusword @bit 8
//     Drive/Inputs/In/nState4 @bit 1 <-> WcState/InputToggle
//     Drive/Inputs/In/nState4 <-> WcState/WcState
//     Drive/Outputs/Out/nCtrl1 <-> Outputs/Controlword
//     Drive/Outputs/Out/nCtrl2 <-> Outputs/Controlword @bit 8
//     Drive/Outputs/Out/nDataOut1 <-> Outputs/Target position
//     Enc/Inputs/In/nDataIn1 <-> Inputs/Position actual value
//     Enc/Inputs/In/nDataIn3 <-> Inputs/Touch probe pos1 pos value
//     Enc/Inputs/In/nDataIn5 <-> Inputs/Touch probe pos2 pos value
//     Enc/Inputs/In/nDcInputTime <-> InfoData/DcInputShift
//     Enc/Inputs/In/nState4 @bit 1 <-> WcState/InputToggle
//     Enc/Inputs/In/nState4 <-> WcState/WcState
//     Enc/Inputs/In/nState5 <-> Inputs/Touch probe status
//     Enc/Inputs/In/nState6 <-> Inputs/Touch probe status @bit 8
//     Enc/Outputs/Out/nCtrl5 <-> Outputs/Touch probe function
//     Enc/Outputs/Out/nCtrl6 <-> Outputs/Touch probe function @bit 8
//   NC-Task 1 SAF/Axes/pm7_buf0 <-> pm side/pm7_buf0
//     Drive/Inputs/In/nDataIn1 <-> Inputs/Following error actual value
//     Drive/Inputs/In/nDataIn3[0] <-> Inputs/Torque actual value
//     Drive/Inputs/In/nDcOutputTime <-> InfoData/DcOutputShift
//     Drive/Inputs/In/nState1 <-> Inputs/Statusword
//     Drive/Inputs/In/nState2 <-> Inputs/Statusword @bit 8
//     Drive/Inputs/In/nState4 @bit 1 <-> WcState/InputToggle
//     Drive/Inputs/In/nState4 <-> WcState/WcState
//     Drive/Outputs/Out/nCtrl1 <-> Outputs/Controlword
//     Drive/Outputs/Out/nCtrl2 <-> Outputs/Controlword @bit 8
//     Drive/Outputs/Out/nDataOut1 <-> Outputs/Target position
//     Enc/Inputs/In/nDataIn1 <-> Inputs/Position actual value
//     Enc/Inputs/In/nDataIn3 <-> Inputs/Touch probe pos1 pos value
//     Enc/Inputs/In/nDataIn5 <-> Inputs/Touch probe pos2 pos value
//     Enc/Inputs/In/nDcInputTime <-> InfoData/DcInputShift
//     Enc/Inputs/In/nState4 @bit 1 <-> WcState/InputToggle
//     Enc/Inputs/In/nState4 <-> WcState/WcState
//     Enc/Inputs/In/nState5 <-> Inputs/Touch probe status
//     Enc/Inputs/In/nState6 <-> Inputs/Touch probe status @bit 8
//     Enc/Outputs/Out/nCtrl5 <-> Outputs/Touch probe function
//     Enc/Outputs/Out/nCtrl6 <-> Outputs/Touch probe function @bit 8
//   NC-Task 1 SAF/Axes/pm7_buf1 <-> pm side/pm7_buf1
//     Drive/Inputs/In/nDataIn1 <-> Inputs/Following error actual value
//     Drive/Inputs/In/nDataIn3[0] <-> Inputs/Torque actual value
//     Drive/Inputs/In/nDcOutputTime <-> InfoData/DcOutputShift
//     Drive/Inputs/In/nState1 <-> Inputs/Statusword
//     Drive/Inputs/In/nState2 <-> Inputs/Statusword @bit 8
//     Drive/Inputs/In/nState4 @bit 1 <-> WcState/InputToggle
//     Drive/Inputs/In/nState4 <-> WcState/WcState
//     Drive/Outputs/Out/nCtrl1 <-> Outputs/Controlword
//     Drive/Outputs/Out/nCtrl2 <-> Outputs/Controlword @bit 8
//     Drive/Outputs/Out/nDataOut1 <-> Outputs/Target position
//     Enc/Inputs/In/nDataIn1 <-> Inputs/Position actual value
//     Enc/Inputs/In/nDataIn3 <-> Inputs/Touch probe pos1 pos value
//     Enc/Inputs/In/nDataIn5 <-> Inputs/Touch probe pos2 pos value
//     Enc/Inputs/In/nDcInputTime <-> InfoData/DcInputShift
//     Enc/Inputs/In/nState4 @bit 1 <-> WcState/InputToggle
//     Enc/Inputs/In/nState4 <-> WcState/WcState
//     Enc/Inputs/In/nState5 <-> Inputs/Touch probe status
//     Enc/Inputs/In/nState6 <-> Inputs/Touch probe status @bit 8
//     Enc/Outputs/Out/nCtrl5 <-> Outputs/Touch probe function
//     Enc/Outputs/Out/nCtrl6 <-> Outputs/Touch probe function @bit 8
//   NC-Task 1 SAF/Axes/pm8_buf0 <-> pm side/pm8_buf0
//     Drive/Inputs/In/nDataIn1 <-> Inputs/Following error actual value
//     Drive/Inputs/In/nDataIn3[0] <-> Inputs/Torque actual value
//     Drive/Inputs/In/nDcOutputTime <-> InfoData/DcOutputShift
//     Drive/Inputs/In/nState1 <-> Inputs/Statusword
//     Drive/Inputs/In/nState2 <-> Inputs/Statusword @bit 8
//     Drive/Inputs/In/nState4 @bit 1 <-> WcState/InputToggle
//     Drive/Inputs/In/nState4 <-> WcState/WcState
//     Drive/Outputs/Out/nCtrl1 <-> Outputs/Controlword
//     Drive/Outputs/Out/nCtrl2 <-> Outputs/Controlword @bit 8
//     Drive/Outputs/Out/nDataOut1 <-> Outputs/Target position
//     Enc/Inputs/In/nDataIn1 <-> Inputs/Position actual value
//     Enc/Inputs/In/nDataIn3 <-> Inputs/Touch probe pos1 pos value
//     Enc/Inputs/In/nDataIn5 <-> Inputs/Touch probe pos2 pos value
//     Enc/Inputs/In/nDcInputTime <-> InfoData/DcInputShift
//     Enc/Inputs/In/nState4 @bit 1 <-> WcState/InputToggle
//     Enc/Inputs/In/nState4 <-> WcState/WcState
//     Enc/Inputs/In/nState5 <-> Inputs/Touch probe status
//     Enc/Inputs/In/nState6 <-> Inputs/Touch probe status @bit 8
//     Enc/Outputs/Out/nCtrl5 <-> Outputs/Touch probe function
//     Enc/Outputs/Out/nCtrl6 <-> Outputs/Touch probe function @bit 8
//   NC-Task 1 SAF/Axes/pm8_buf1 <-> pm side/pm8_buf1
//     Drive/Inputs/In/nDataIn1 <-> Inputs/Following error actual value
//     Drive/Inputs/In/nDataIn3[0] <-> Inputs/Torque actual value
//     Drive/Inputs/In/nDcOutputTime <-> InfoData/DcOutputShift
//     Drive/Inputs/In/nState1 <-> Inputs/Statusword
//     Drive/Inputs/In/nState2 <-> Inputs/Statusword @bit 8
//     Drive/Inputs/In/nState4 @bit 1 <-> WcState/InputToggle
//     Drive/Inputs/In/nState4 <-> WcState/WcState
//     Drive/Outputs/Out/nCtrl1 <-> Outputs/Controlword
//     Drive/Outputs/Out/nCtrl2 <-> Outputs/Controlword @bit 8
//     Drive/Outputs/Out/nDataOut1 <-> Outputs/Target position
//     Enc/Inputs/In/nDataIn1 <-> Inputs/Position actual value
//     Enc/Inputs/In/nDataIn3 <-> Inputs/Touch probe pos1 pos value
//     Enc/Inputs/In/nDataIn5 <-> Inputs/Touch probe pos2 pos value
//     Enc/Inputs/In/nDcInputTime <-> InfoData/DcInputShift
//     Enc/Inputs/In/nState4 @bit 1 <-> WcState/InputToggle
//     Enc/Inputs/In/nState4 <-> WcState/WcState
//     Enc/Inputs/In/nState5 <-> Inputs/Touch probe status
//     Enc/Inputs/In/nState6 <-> Inputs/Touch probe status @bit 8
//     Enc/Outputs/Out/nCtrl5 <-> Outputs/Touch probe function
//     Enc/Outputs/Out/nCtrl6 <-> Outputs/Touch probe function @bit 8
//   NC-Task 1 SAF/Axes/pm9_buf0 <-> pm side/pm9_buf0
//     Drive/Inputs/In/nDataIn1 <-> Inputs/Following error actual value
//     Drive/Inputs/In/nDataIn3[0] <-> Inputs/Torque actual value
//     Drive/Inputs/In/nDcOutputTime <-> InfoData/DcOutputShift
//     Drive/Inputs/In/nState1 <-> Inputs/Statusword
//     Drive/Inputs/In/nState2 <-> Inputs/Statusword @bit 8
//     Drive/Inputs/In/nState4 @bit 1 <-> WcState/InputToggle
//     Drive/Inputs/In/nState4 <-> WcState/WcState
//     Drive/Outputs/Out/nCtrl1 <-> Outputs/Controlword
//     Drive/Outputs/Out/nCtrl2 <-> Outputs/Controlword @bit 8
//     Drive/Outputs/Out/nDataOut1 <-> Outputs/Target position
//     Enc/Inputs/In/nDataIn1 <-> Inputs/Position actual value
//     Enc/Inputs/In/nDataIn3 <-> Inputs/Touch probe pos1 pos value
//     Enc/Inputs/In/nDataIn5 <-> Inputs/Touch probe pos2 pos value
//     Enc/Inputs/In/nDcInputTime <-> InfoData/DcInputShift
//     Enc/Inputs/In/nState4 @bit 1 <-> WcState/InputToggle
//     Enc/Inputs/In/nState4 <-> WcState/WcState
//     Enc/Inputs/In/nState5 <-> Inputs/Touch probe status
//     Enc/Inputs/In/nState6 <-> Inputs/Touch probe status @bit 8
//     Enc/Outputs/Out/nCtrl5 <-> Outputs/Touch probe function
//     Enc/Outputs/Out/nCtrl6 <-> Outputs/Touch probe function @bit 8
//   NC-Task 1 SAF/Axes/pm9_buf1 <-> pm side/pm9_buf1
//     Drive/Inputs/In/nDataIn1 <-> Inputs/Following error actual value
//     Drive/Inputs/In/nDataIn3[0] <-> Inputs/Torque actual value
//     Drive/Inputs/In/nDcOutputTime <-> InfoData/DcOutputShift
//     Drive/Inputs/In/nState1 <-> Inputs/Statusword
//     Drive/Inputs/In/nState2 <-> Inputs/Statusword @bit 8
//     Drive/Inputs/In/nState4 @bit 1 <-> WcState/InputToggle
//     Drive/Inputs/In/nState4 <-> WcState/WcState
//     Drive/Outputs/Out/nCtrl1 <-> Outputs/Controlword
//     Drive/Outputs/Out/nCtrl2 <-> Outputs/Controlword @bit 8
//     Drive/Outputs/Out/nDataOut1 <-> Outputs/Target position
//     Enc/Inputs/In/nDataIn1 <-> Inputs/Position actual value
//     Enc/Inputs/In/nDataIn3 <-> Inputs/Touch probe pos1 pos value
//     Enc/Inputs/In/nDataIn5 <-> Inputs/Touch probe pos2 pos value
//     Enc/Inputs/In/nDcInputTime <-> InfoData/DcInputShift
//     Enc/Inputs/In/nState4 @bit 1 <-> WcState/InputToggle
//     Enc/Inputs/In/nState4 <-> WcState/WcState
//     Enc/Inputs/In/nState5 <-> Inputs/Touch probe status
//     Enc/Inputs/In/nState6 <-> Inputs/Touch probe status @bit 8
//     Enc/Outputs/Out/nCtrl5 <-> Outputs/Touch probe function
//     Enc/Outputs/Out/nCtrl6 <-> Outputs/Touch probe function @bit 8
//   NC-Task 1 SAF/Axes/rem0_Lift0 <-> rem_wf/rem0_Lift0
//     Drive/Inputs/In/nDataIn1 <-> Inputs/Following error actual value
//     Drive/Inputs/In/nDataIn3[0] <-> Inputs/Torque actual value
//     Drive/Inputs/In/nDcOutputTime <-> InfoData/DcOutputShift
//     Drive/Inputs/In/nState1 <-> Inputs/Statusword
//     Drive/Inputs/In/nState2 <-> Inputs/Statusword @bit 8
//     Drive/Inputs/In/nState4 @bit 1 <-> WcState/InputToggle
//     Drive/Inputs/In/nState4 <-> WcState/WcState
//     Drive/Outputs/Out/nCtrl1 <-> Outputs/Controlword
//     Drive/Outputs/Out/nCtrl2 <-> Outputs/Controlword @bit 8
//     Drive/Outputs/Out/nDataOut1 <-> Outputs/Target position
//     Enc/Inputs/In/nDataIn1 <-> Inputs/Position actual value
//     Enc/Inputs/In/nDataIn3 <-> Inputs/Touch probe pos1 pos value
//     Enc/Inputs/In/nDataIn5 <-> Inputs/Touch probe pos2 pos value
//     Enc/Inputs/In/nDcInputTime <-> InfoData/DcInputShift
//     Enc/Inputs/In/nState4 @bit 1 <-> WcState/InputToggle
//     Enc/Inputs/In/nState4 <-> WcState/WcState
//     Enc/Inputs/In/nState5 <-> Inputs/Touch probe status
//     Enc/Inputs/In/nState6 <-> Inputs/Touch probe status @bit 8
//     Enc/Outputs/Out/nCtrl5 <-> Outputs/Touch probe function
//     Enc/Outputs/Out/nCtrl6 <-> Outputs/Touch probe function @bit 8
//   NC-Task 1 SAF/Axes/rem0_Lift1 <-> rem_wf/rem0_Lift1
//     Drive/Inputs/In/nDataIn1 <-> Inputs/Following error actual value
//     Drive/Inputs/In/nDataIn3[0] <-> Inputs/Torque actual value
//     Drive/Inputs/In/nDcOutputTime <-> InfoData/DcOutputShift
//     Drive/Inputs/In/nState1 <-> Inputs/Statusword
//     Drive/Inputs/In/nState2 <-> Inputs/Statusword @bit 8
//     Drive/Inputs/In/nState4 @bit 1 <-> WcState/InputToggle
//     Drive/Inputs/In/nState4 <-> WcState/WcState
//     Drive/Outputs/Out/nCtrl1 <-> Outputs/Controlword
//     Drive/Outputs/Out/nCtrl2 <-> Outputs/Controlword @bit 8
//     Drive/Outputs/Out/nDataOut1 <-> Outputs/Target position
//     Enc/Inputs/In/nDataIn1 <-> Inputs/Position actual value
//     Enc/Inputs/In/nDataIn3 <-> Inputs/Touch probe pos1 pos value
//     Enc/Inputs/In/nDataIn5 <-> Inputs/Touch probe pos2 pos value
//     Enc/Inputs/In/nDcInputTime <-> InfoData/DcInputShift
//     Enc/Inputs/In/nState4 @bit 1 <-> WcState/InputToggle
//     Enc/Inputs/In/nState4 <-> WcState/WcState
//     Enc/Inputs/In/nState5 <-> Inputs/Touch probe status
//     Enc/Inputs/In/nState6 <-> Inputs/Touch probe status @bit 8
//     Enc/Outputs/Out/nCtrl5 <-> Outputs/Touch probe function
//     Enc/Outputs/Out/nCtrl6 <-> Outputs/Touch probe function @bit 8
//   NC-Task 1 SAF/Axes/rem1_Lift0 <-> rem_wf/rem1_Lift0
//     Drive/Inputs/In/nDataIn1 <-> Inputs/Following error actual value
//     Drive/Inputs/In/nDataIn3[0] <-> Inputs/Torque actual value
//     Drive/Inputs/In/nDcOutputTime <-> InfoData/DcOutputShift
//     Drive/Inputs/In/nState1 <-> Inputs/Statusword
//     Drive/Inputs/In/nState2 <-> Inputs/Statusword @bit 8
//     Drive/Inputs/In/nState4 @bit 1 <-> WcState/InputToggle
//     Drive/Inputs/In/nState4 <-> WcState/WcState
//     Drive/Outputs/Out/nCtrl1 <-> Outputs/Controlword
//     Drive/Outputs/Out/nCtrl2 <-> Outputs/Controlword @bit 8
//     Drive/Outputs/Out/nDataOut1 <-> Outputs/Target position
//     Enc/Inputs/In/nDataIn1 <-> Inputs/Position actual value
//     Enc/Inputs/In/nDataIn3 <-> Inputs/Touch probe pos1 pos value
//     Enc/Inputs/In/nDataIn5 <-> Inputs/Touch probe pos2 pos value
//     Enc/Inputs/In/nDcInputTime <-> InfoData/DcInputShift
//     Enc/Inputs/In/nState4 @bit 1 <-> WcState/InputToggle
//     Enc/Inputs/In/nState4 <-> WcState/WcState
//     Enc/Inputs/In/nState5 <-> Inputs/Touch probe status
//     Enc/Inputs/In/nState6 <-> Inputs/Touch probe status @bit 8
//     Enc/Outputs/Out/nCtrl5 <-> Outputs/Touch probe function
//     Enc/Outputs/Out/nCtrl6 <-> Outputs/Touch probe function @bit 8
//   NC-Task 1 SAF/Axes/rem1_Lift1 <-> rem_wf/rem1_Lift1
//     Drive/Inputs/In/nDataIn1 <-> Inputs/Following error actual value
//     Drive/Inputs/In/nDataIn3[0] <-> Inputs/Torque actual value
//     Drive/Inputs/In/nDcOutputTime <-> InfoData/DcOutputShift
//     Drive/Inputs/In/nState1 <-> Inputs/Statusword
//     Drive/Inputs/In/nState2 <-> Inputs/Statusword @bit 8
//     Drive/Inputs/In/nState4 @bit 1 <-> WcState/InputToggle
//     Drive/Inputs/In/nState4 <-> WcState/WcState
//     Drive/Outputs/Out/nCtrl1 <-> Outputs/Controlword
//     Drive/Outputs/Out/nCtrl2 <-> Outputs/Controlword @bit 8
//     Drive/Outputs/Out/nDataOut1 <-> Outputs/Target position
//     Enc/Inputs/In/nDataIn1 <-> Inputs/Position actual value
//     Enc/Inputs/In/nDataIn3 <-> Inputs/Touch probe pos1 pos value
//     Enc/Inputs/In/nDataIn5 <-> Inputs/Touch probe pos2 pos value
//     Enc/Inputs/In/nDcInputTime <-> InfoData/DcInputShift
//     Enc/Inputs/In/nState4 @bit 1 <-> WcState/InputToggle
//     Enc/Inputs/In/nState4 <-> WcState/WcState
//     Enc/Inputs/In/nState5 <-> Inputs/Touch probe status
//     Enc/Inputs/In/nState6 <-> Inputs/Touch probe status @bit 8
//     Enc/Outputs/Out/nCtrl5 <-> Outputs/Touch probe function
//     Enc/Outputs/Out/nCtrl6 <-> Outputs/Touch probe function @bit 8
//   NC-Task 1 SAF/Axes/rem2_Lift0 <-> rem_wf/rem2_Lift0
//     Drive/Inputs/In/nDataIn1 <-> Inputs/Following error actual value
//     Drive/Inputs/In/nDataIn3[0] <-> Inputs/Torque actual value
//     Drive/Inputs/In/nDcOutputTime <-> InfoData/DcOutputShift
//     Drive/Inputs/In/nState1 <-> Inputs/Statusword
//     Drive/Inputs/In/nState2 <-> Inputs/Statusword @bit 8
//     Drive/Inputs/In/nState4 @bit 1 <-> WcState/InputToggle
//     Drive/Inputs/In/nState4 <-> WcState/WcState
//     Drive/Outputs/Out/nCtrl1 <-> Outputs/Controlword
//     Drive/Outputs/Out/nCtrl2 <-> Outputs/Controlword @bit 8
//     Drive/Outputs/Out/nDataOut1 <-> Outputs/Target position
//     Enc/Inputs/In/nDataIn1 <-> Inputs/Position actual value
//     Enc/Inputs/In/nDataIn3 <-> Inputs/Touch probe pos1 pos value
//     Enc/Inputs/In/nDataIn5 <-> Inputs/Touch probe pos2 pos value
//     Enc/Inputs/In/nDcInputTime <-> InfoData/DcInputShift
//     Enc/Inputs/In/nState4 @bit 1 <-> WcState/InputToggle
//     Enc/Inputs/In/nState4 <-> WcState/WcState
//     Enc/Inputs/In/nState5 <-> Inputs/Touch probe status
//     Enc/Inputs/In/nState6 <-> Inputs/Touch probe status @bit 8
//     Enc/Outputs/Out/nCtrl5 <-> Outputs/Touch probe function
//     Enc/Outputs/Out/nCtrl6 <-> Outputs/Touch probe function @bit 8
//   NC-Task 1 SAF/Axes/rem2_Lift1 <-> rem_wf/rem2_Lift1
//     Drive/Inputs/In/nDataIn1 <-> Inputs/Following error actual value
//     Drive/Inputs/In/nDataIn3[0] <-> Inputs/Torque actual value
//     Drive/Inputs/In/nDcOutputTime <-> InfoData/DcOutputShift
//     Drive/Inputs/In/nState1 <-> Inputs/Statusword
//     Drive/Inputs/In/nState2 <-> Inputs/Statusword @bit 8
//     Drive/Inputs/In/nState4 @bit 1 <-> WcState/InputToggle
//     Drive/Inputs/In/nState4 <-> WcState/WcState
//     Drive/Outputs/Out/nCtrl1 <-> Outputs/Controlword
//     Drive/Outputs/Out/nCtrl2 <-> Outputs/Controlword @bit 8
//     Drive/Outputs/Out/nDataOut1 <-> Outputs/Target position
//     Enc/Inputs/In/nDataIn1 <-> Inputs/Position actual value
//     Enc/Inputs/In/nDataIn3 <-> Inputs/Touch probe pos1 pos value
//     Enc/Inputs/In/nDataIn5 <-> Inputs/Touch probe pos2 pos value
//     Enc/Inputs/In/nDcInputTime <-> InfoData/DcInputShift
//     Enc/Inputs/In/nState4 @bit 1 <-> WcState/InputToggle
//     Enc/Inputs/In/nState4 <-> WcState/WcState
//     Enc/Inputs/In/nState5 <-> Inputs/Touch probe status
//     Enc/Inputs/In/nState6 <-> Inputs/Touch probe status @bit 8
//     Enc/Outputs/Out/nCtrl5 <-> Outputs/Touch probe function
//     Enc/Outputs/Out/nCtrl6 <-> Outputs/Touch probe function @bit 8
//   NC-Task 1 SAF/Axes/rem3_Lift0 <-> rem_wf/rem3_Lift0
//     Drive/Inputs/In/nDataIn1 <-> Inputs/Following error actual value
//     Drive/Inputs/In/nDataIn3[0] <-> Inputs/Torque actual value
//     Drive/Inputs/In/nDcOutputTime <-> InfoData/DcOutputShift
//     Drive/Inputs/In/nState1 <-> Inputs/Statusword
//     Drive/Inputs/In/nState2 <-> Inputs/Statusword @bit 8
//     Drive/Inputs/In/nState4 @bit 1 <-> WcState/InputToggle
//     Drive/Inputs/In/nState4 <-> WcState/WcState
//     Drive/Outputs/Out/nCtrl1 <-> Outputs/Controlword
//     Drive/Outputs/Out/nCtrl2 <-> Outputs/Controlword @bit 8
//     Drive/Outputs/Out/nDataOut1 <-> Outputs/Target position
//     Enc/Inputs/In/nDataIn1 <-> Inputs/Position actual value
//     Enc/Inputs/In/nDataIn3 <-> Inputs/Touch probe pos1 pos value
//     Enc/Inputs/In/nDataIn5 <-> Inputs/Touch probe pos2 pos value
//     Enc/Inputs/In/nDcInputTime <-> InfoData/DcInputShift
//     Enc/Inputs/In/nState4 @bit 1 <-> WcState/InputToggle
//     Enc/Inputs/In/nState4 <-> WcState/WcState
//     Enc/Inputs/In/nState5 <-> Inputs/Touch probe status
//     Enc/Inputs/In/nState6 <-> Inputs/Touch probe status @bit 8
//     Enc/Outputs/Out/nCtrl5 <-> Outputs/Touch probe function
//     Enc/Outputs/Out/nCtrl6 <-> Outputs/Touch probe function @bit 8
//   NC-Task 1 SAF/Axes/rem3_Lift1 <-> rem_wf/rem3_Lift1
//     Drive/Inputs/In/nDataIn1 <-> Inputs/Following error actual value
//     Drive/Inputs/In/nDataIn3[0] <-> Inputs/Torque actual value
//     Drive/Inputs/In/nDcOutputTime <-> InfoData/DcOutputShift
//     Drive/Inputs/In/nState1 <-> Inputs/Statusword
//     Drive/Inputs/In/nState2 <-> Inputs/Statusword @bit 8
//     Drive/Inputs/In/nState4 @bit 1 <-> WcState/InputToggle
//     Drive/Inputs/In/nState4 <-> WcState/WcState
//     Drive/Outputs/Out/nCtrl1 <-> Outputs/Controlword
//     Drive/Outputs/Out/nCtrl2 <-> Outputs/Controlword @bit 8
//     Drive/Outputs/Out/nDataOut1 <-> Outputs/Target position
//     Enc/Inputs/In/nDataIn1 <-> Inputs/Position actual value
//     Enc/Inputs/In/nDataIn3 <-> Inputs/Touch probe pos1 pos value
//     Enc/Inputs/In/nDataIn5 <-> Inputs/Touch probe pos2 pos value
//     Enc/Inputs/In/nDcInputTime <-> InfoData/DcInputShift
//     Enc/Inputs/In/nState4 @bit 1 <-> WcState/InputToggle
//     Enc/Inputs/In/nState4 <-> WcState/WcState
//     Enc/Inputs/In/nState5 <-> Inputs/Touch probe status
//     Enc/Inputs/In/nState6 <-> Inputs/Touch probe status @bit 8
//     Enc/Outputs/Out/nCtrl5 <-> Outputs/Touch probe function
//     Enc/Outputs/Out/nCtrl6 <-> Outputs/Touch probe function @bit 8
//   NC-Task 1 SAF/Axes/rem4_Lift0 <-> rem_wf/rem4_Lift0
//     Drive/Inputs/In/nDataIn1 <-> Inputs/Following error actual value
//     Drive/Inputs/In/nDataIn3[0] <-> Inputs/Torque actual value
//     Drive/Inputs/In/nDcOutputTime <-> InfoData/DcOutputShift
//     Drive/Inputs/In/nState1 <-> Inputs/Statusword
//     Drive/Inputs/In/nState2 <-> Inputs/Statusword @bit 8
//     Drive/Inputs/In/nState4 @bit 1 <-> WcState/InputToggle
//     Drive/Inputs/In/nState4 <-> WcState/WcState
//     Drive/Outputs/Out/nCtrl1 <-> Outputs/Controlword
//     Drive/Outputs/Out/nCtrl2 <-> Outputs/Controlword @bit 8
//     Drive/Outputs/Out/nDataOut1 <-> Outputs/Target position
//     Enc/Inputs/In/nDataIn1 <-> Inputs/Position actual value
//     Enc/Inputs/In/nDataIn3 <-> Inputs/Touch probe pos1 pos value
//     Enc/Inputs/In/nDataIn5 <-> Inputs/Touch probe pos2 pos value
//     Enc/Inputs/In/nDcInputTime <-> InfoData/DcInputShift
//     Enc/Inputs/In/nState4 @bit 1 <-> WcState/InputToggle
//     Enc/Inputs/In/nState4 <-> WcState/WcState
//     Enc/Inputs/In/nState5 <-> Inputs/Touch probe status
//     Enc/Inputs/In/nState6 <-> Inputs/Touch probe status @bit 8
//     Enc/Outputs/Out/nCtrl5 <-> Outputs/Touch probe function
//     Enc/Outputs/Out/nCtrl6 <-> Outputs/Touch probe function @bit 8
//   NC-Task 1 SAF/Axes/rem4_Lift1 <-> rem_wf/rem4_Lift1
//     Drive/Inputs/In/nDataIn1 <-> Inputs/Following error actual value
//     Drive/Inputs/In/nDataIn3[0] <-> Inputs/Torque actual value
//     Drive/Inputs/In/nDcOutputTime <-> InfoData/DcOutputShift
//     Drive/Inputs/In/nState1 <-> Inputs/Statusword
//     Drive/Inputs/In/nState2 <-> Inputs/Statusword @bit 8
//     Drive/Inputs/In/nState4 @bit 1 <-> WcState/InputToggle
//     Drive/Inputs/In/nState4 <-> WcState/WcState
//     Drive/Outputs/Out/nCtrl1 <-> Outputs/Controlword
//     Drive/Outputs/Out/nCtrl2 <-> Outputs/Controlword @bit 8
//     Drive/Outputs/Out/nDataOut1 <-> Outputs/Target position
//     Enc/Inputs/In/nDataIn1 <-> Inputs/Position actual value
//     Enc/Inputs/In/nDataIn3 <-> Inputs/Touch probe pos1 pos value
//     Enc/Inputs/In/nDataIn5 <-> Inputs/Touch probe pos2 pos value
//     Enc/Inputs/In/nDcInputTime <-> InfoData/DcInputShift
//     Enc/Inputs/In/nState4 @bit 1 <-> WcState/InputToggle
//     Enc/Inputs/In/nState4 <-> WcState/WcState
//     Enc/Inputs/In/nState5 <-> Inputs/Touch probe status
//     Enc/Inputs/In/nState6 <-> Inputs/Touch probe status @bit 8
//     Enc/Outputs/Out/nCtrl5 <-> Outputs/Touch probe function
//     Enc/Outputs/Out/nCtrl6 <-> Outputs/Touch probe function @bit 8
//   NC-Task 1 SAF/Axes/rem5_Lift0 <-> rem_wf/rem5_Lift0
//     Drive/Inputs/In/nDataIn1 <-> Inputs/Following error actual value
//     Drive/Inputs/In/nDataIn3[0] <-> Inputs/Torque actual value
//     Drive/Inputs/In/nDcOutputTime <-> InfoData/DcOutputShift
//     Drive/Inputs/In/nState1 <-> Inputs/Statusword
//     Drive/Inputs/In/nState2 <-> Inputs/Statusword @bit 8
//     Drive/Inputs/In/nState4 @bit 1 <-> WcState/InputToggle
//     Drive/Inputs/In/nState4 <-> WcState/WcState
//     Drive/Outputs/Out/nCtrl1 <-> Outputs/Controlword
//     Drive/Outputs/Out/nCtrl2 <-> Outputs/Controlword @bit 8
//     Drive/Outputs/Out/nDataOut1 <-> Outputs/Target position
//     Enc/Inputs/In/nDataIn1 <-> Inputs/Position actual value
//     Enc/Inputs/In/nDataIn3 <-> Inputs/Touch probe pos1 pos value
//     Enc/Inputs/In/nDataIn5 <-> Inputs/Touch probe pos2 pos value
//     Enc/Inputs/In/nDcInputTime <-> InfoData/DcInputShift
//     Enc/Inputs/In/nState4 @bit 1 <-> WcState/InputToggle
//     Enc/Inputs/In/nState4 <-> WcState/WcState
//     Enc/Inputs/In/nState5 <-> Inputs/Touch probe status
//     Enc/Inputs/In/nState6 <-> Inputs/Touch probe status @bit 8
//     Enc/Outputs/Out/nCtrl5 <-> Outputs/Touch probe function
//     Enc/Outputs/Out/nCtrl6 <-> Outputs/Touch probe function @bit 8
//   NC-Task 1 SAF/Axes/rem5_Lift1 <-> rem_wf/rem5_Lift1
//     Drive/Inputs/In/nDataIn1 <-> Inputs/Following error actual value
//     Drive/Inputs/In/nDataIn3[0] <-> Inputs/Torque actual value
//     Drive/Inputs/In/nDcOutputTime <-> InfoData/DcOutputShift
//     Drive/Inputs/In/nState1 <-> Inputs/Statusword
//     Drive/Inputs/In/nState2 <-> Inputs/Statusword @bit 8
//     Drive/Inputs/In/nState4 @bit 1 <-> WcState/InputToggle
//     Drive/Inputs/In/nState4 <-> WcState/WcState
//     Drive/Outputs/Out/nCtrl1 <-> Outputs/Controlword
//     Drive/Outputs/Out/nCtrl2 <-> Outputs/Controlword @bit 8
//     Drive/Outputs/Out/nDataOut1 <-> Outputs/Target position
//     Enc/Inputs/In/nDataIn1 <-> Inputs/Position actual value
//     Enc/Inputs/In/nDataIn3 <-> Inputs/Touch probe pos1 pos value
//     Enc/Inputs/In/nDataIn5 <-> Inputs/Touch probe pos2 pos value
//     Enc/Inputs/In/nDcInputTime <-> InfoData/DcInputShift
//     Enc/Inputs/In/nState4 @bit 1 <-> WcState/InputToggle
//     Enc/Inputs/In/nState4 <-> WcState/WcState
//     Enc/Inputs/In/nState5 <-> Inputs/Touch probe status
//     Enc/Inputs/In/nState6 <-> Inputs/Touch probe status @bit 8
//     Enc/Outputs/Out/nCtrl5 <-> Outputs/Touch probe function
//     Enc/Outputs/Out/nCtrl6 <-> Outputs/Touch probe function @bit 8
//   NC-Task 1 SAF/Axes/rem6_Lift0 <-> rem_wf/rem6_Lift0
//     Drive/Inputs/In/nDataIn1 <-> Inputs/Following error actual value
//     Drive/Inputs/In/nDataIn3[0] <-> Inputs/Torque actual value
//     Drive/Inputs/In/nDcOutputTime <-> InfoData/DcOutputShift
//     Drive/Inputs/In/nState1 <-> Inputs/Statusword
//     Drive/Inputs/In/nState2 <-> Inputs/Statusword @bit 8
//     Drive/Inputs/In/nState4 @bit 1 <-> WcState/InputToggle
//     Drive/Inputs/In/nState4 <-> WcState/WcState
//     Drive/Outputs/Out/nCtrl1 <-> Outputs/Controlword
//     Drive/Outputs/Out/nCtrl2 <-> Outputs/Controlword @bit 8
//     Drive/Outputs/Out/nDataOut1 <-> Outputs/Target position
//     Enc/Inputs/In/nDataIn1 <-> Inputs/Position actual value
//     Enc/Inputs/In/nDataIn3 <-> Inputs/Touch probe pos1 pos value
//     Enc/Inputs/In/nDataIn5 <-> Inputs/Touch probe pos2 pos value
//     Enc/Inputs/In/nDcInputTime <-> InfoData/DcInputShift
//     Enc/Inputs/In/nState4 @bit 1 <-> WcState/InputToggle
//     Enc/Inputs/In/nState4 <-> WcState/WcState
//     Enc/Inputs/In/nState5 <-> Inputs/Touch probe status
//     Enc/Inputs/In/nState6 <-> Inputs/Touch probe status @bit 8
//     Enc/Outputs/Out/nCtrl5 <-> Outputs/Touch probe function
//     Enc/Outputs/Out/nCtrl6 <-> Outputs/Touch probe function @bit 8
//   NC-Task 1 SAF/Axes/rem6_Lift1 <-> rem_wf/rem6_Lift1
//     Drive/Inputs/In/nDataIn1 <-> Inputs/Following error actual value
//     Drive/Inputs/In/nDataIn3[0] <-> Inputs/Torque actual value
//     Drive/Inputs/In/nDcOutputTime <-> InfoData/DcOutputShift
//     Drive/Inputs/In/nState1 <-> Inputs/Statusword
//     Drive/Inputs/In/nState2 <-> Inputs/Statusword @bit 8
//     Drive/Inputs/In/nState4 @bit 1 <-> WcState/InputToggle
//     Drive/Inputs/In/nState4 <-> WcState/WcState
//     Drive/Outputs/Out/nCtrl1 <-> Outputs/Controlword
//     Drive/Outputs/Out/nCtrl2 <-> Outputs/Controlword @bit 8
//     Drive/Outputs/Out/nDataOut1 <-> Outputs/Target position
//     Enc/Inputs/In/nDataIn1 <-> Inputs/Position actual value
//     Enc/Inputs/In/nDataIn3 <-> Inputs/Touch probe pos1 pos value
//     Enc/Inputs/In/nDataIn5 <-> Inputs/Touch probe pos2 pos value
//     Enc/Inputs/In/nDcInputTime <-> InfoData/DcInputShift
//     Enc/Inputs/In/nState4 @bit 1 <-> WcState/InputToggle
//     Enc/Inputs/In/nState4 <-> WcState/WcState
//     Enc/Inputs/In/nState5 <-> Inputs/Touch probe status
//     Enc/Inputs/In/nState6 <-> Inputs/Touch probe status @bit 8
//     Enc/Outputs/Out/nCtrl5 <-> Outputs/Touch probe function
//     Enc/Outputs/Out/nCtrl6 <-> Outputs/Touch probe function @bit 8
//   NC-Task 1 SAF/Axes/rem7_Lift0 <-> rem_wf/rem7_Lift0
//     Drive/Inputs/In/nDataIn1 <-> Inputs/Following error actual value
//     Drive/Inputs/In/nDataIn3[0] <-> Inputs/Torque actual value
//     Drive/Inputs/In/nDcOutputTime <-> InfoData/DcOutputShift
//     Drive/Inputs/In/nState1 <-> Inputs/Statusword
//     Drive/Inputs/In/nState2 <-> Inputs/Statusword @bit 8
//     Drive/Inputs/In/nState4 @bit 1 <-> WcState/InputToggle
//     Drive/Inputs/In/nState4 <-> WcState/WcState
//     Drive/Outputs/Out/nCtrl1 <-> Outputs/Controlword
//     Drive/Outputs/Out/nCtrl2 <-> Outputs/Controlword @bit 8
//     Drive/Outputs/Out/nDataOut1 <-> Outputs/Target position
//     Enc/Inputs/In/nDataIn1 <-> Inputs/Position actual value
//     Enc/Inputs/In/nDataIn3 <-> Inputs/Touch probe pos1 pos value
//     Enc/Inputs/In/nDataIn5 <-> Inputs/Touch probe pos2 pos value
//     Enc/Inputs/In/nDcInputTime <-> InfoData/DcInputShift
//     Enc/Inputs/In/nState4 @bit 1 <-> WcState/InputToggle
//     Enc/Inputs/In/nState4 <-> WcState/WcState
//     Enc/Inputs/In/nState5 <-> Inputs/Touch probe status
//     Enc/Inputs/In/nState6 <-> Inputs/Touch probe status @bit 8
//     Enc/Outputs/Out/nCtrl5 <-> Outputs/Touch probe function
//     Enc/Outputs/Out/nCtrl6 <-> Outputs/Touch probe function @bit 8
//   NC-Task 1 SAF/Axes/rem7_Lift1 <-> rem_wf/rem7_Lift1
//     Drive/Inputs/In/nDataIn1 <-> Inputs/Following error actual value
//     Drive/Inputs/In/nDataIn3[0] <-> Inputs/Torque actual value
//     Drive/Inputs/In/nDcOutputTime <-> InfoData/DcOutputShift
//     Drive/Inputs/In/nState1 <-> Inputs/Statusword
//     Drive/Inputs/In/nState2 <-> Inputs/Statusword @bit 8
//     Drive/Inputs/In/nState4 @bit 1 <-> WcState/InputToggle
//     Drive/Inputs/In/nState4 <-> WcState/WcState
//     Drive/Outputs/Out/nCtrl1 <-> Outputs/Controlword
//     Drive/Outputs/Out/nCtrl2 <-> Outputs/Controlword @bit 8
//     Drive/Outputs/Out/nDataOut1 <-> Outputs/Target position
//     Enc/Inputs/In/nDataIn1 <-> Inputs/Position actual value
//     Enc/Inputs/In/nDataIn3 <-> Inputs/Touch probe pos1 pos value
//     Enc/Inputs/In/nDataIn5 <-> Inputs/Touch probe pos2 pos value
//     Enc/Inputs/In/nDcInputTime <-> InfoData/DcInputShift
//     Enc/Inputs/In/nState4 @bit 1 <-> WcState/InputToggle
//     Enc/Inputs/In/nState4 <-> WcState/WcState
//     Enc/Inputs/In/nState5 <-> Inputs/Touch probe status
//     Enc/Inputs/In/nState6 <-> Inputs/Touch probe status @bit 8
//     Enc/Outputs/Out/nCtrl5 <-> Outputs/Touch probe function
//     Enc/Outputs/Out/nCtrl6 <-> Outputs/Touch probe function @bit 8
//   NC-Task 1 SAF/Axes/rem8_Lift0 <-> rem_wf/rem8_Lift0
//     Drive/Inputs/In/nDataIn1 <-> Inputs/Following error actual value
//     Drive/Inputs/In/nDataIn3[0] <-> Inputs/Torque actual value
//     Drive/Inputs/In/nDcOutputTime <-> InfoData/DcOutputShift
//     Drive/Inputs/In/nState1 <-> Inputs/Statusword
//     Drive/Inputs/In/nState2 <-> Inputs/Statusword @bit 8
//     Drive/Inputs/In/nState4 @bit 1 <-> WcState/InputToggle
//     Drive/Inputs/In/nState4 <-> WcState/WcState
//     Drive/Outputs/Out/nCtrl1 <-> Outputs/Controlword
//     Drive/Outputs/Out/nCtrl2 <-> Outputs/Controlword @bit 8
//     Drive/Outputs/Out/nDataOut1 <-> Outputs/Target position
//     Enc/Inputs/In/nDataIn1 <-> Inputs/Position actual value
//     Enc/Inputs/In/nDataIn3 <-> Inputs/Touch probe pos1 pos value
//     Enc/Inputs/In/nDataIn5 <-> Inputs/Touch probe pos2 pos value
//     Enc/Inputs/In/nDcInputTime <-> InfoData/DcInputShift
//     Enc/Inputs/In/nState4 @bit 1 <-> WcState/InputToggle
//     Enc/Inputs/In/nState4 <-> WcState/WcState
//     Enc/Inputs/In/nState5 <-> Inputs/Touch probe status
//     Enc/Inputs/In/nState6 <-> Inputs/Touch probe status @bit 8
//     Enc/Outputs/Out/nCtrl5 <-> Outputs/Touch probe function
//     Enc/Outputs/Out/nCtrl6 <-> Outputs/Touch probe function @bit 8
//   NC-Task 1 SAF/Axes/rem8_Lift1 <-> rem_wf/rem8_Lift1
//     Drive/Inputs/In/nDataIn1 <-> Inputs/Following error actual value
//     Drive/Inputs/In/nDataIn3[0] <-> Inputs/Torque actual value
//     Drive/Inputs/In/nDcOutputTime <-> InfoData/DcOutputShift
//     Drive/Inputs/In/nState1 <-> Inputs/Statusword
//     Drive/Inputs/In/nState2 <-> Inputs/Statusword @bit 8
//     Drive/Inputs/In/nState4 @bit 1 <-> WcState/InputToggle
//     Drive/Inputs/In/nState4 <-> WcState/WcState
//     Drive/Outputs/Out/nCtrl1 <-> Outputs/Controlword
//     Drive/Outputs/Out/nCtrl2 <-> Outputs/Controlword @bit 8
//     Drive/Outputs/Out/nDataOut1 <-> Outputs/Target position
//     Enc/Inputs/In/nDataIn1 <-> Inputs/Position actual value
//     Enc/Inputs/In/nDataIn3 <-> Inputs/Touch probe pos1 pos value
//     Enc/Inputs/In/nDataIn5 <-> Inputs/Touch probe pos2 pos value
//     Enc/Inputs/In/nDcInputTime <-> InfoData/DcInputShift
//     Enc/Inputs/In/nState4 @bit 1 <-> WcState/InputToggle
//     Enc/Inputs/In/nState4 <-> WcState/WcState
//     Enc/Inputs/In/nState5 <-> Inputs/Touch probe status
//     Enc/Inputs/In/nState6 <-> Inputs/Touch probe status @bit 8
//     Enc/Outputs/Out/nCtrl5 <-> Outputs/Touch probe function
//     Enc/Outputs/Out/nCtrl6 <-> Outputs/Touch probe function @bit 8
//   NC-Task 1 SAF/Axes/rem9_Lift0 <-> rem_wf/rem9_Lift0
//     Drive/Inputs/In/nDataIn1 <-> Inputs/Following error actual value
//     Drive/Inputs/In/nDataIn3[0] <-> Inputs/Torque actual value
//     Drive/Inputs/In/nDcOutputTime <-> InfoData/DcOutputShift
//     Drive/Inputs/In/nState1 <-> Inputs/Statusword
//     Drive/Inputs/In/nState2 <-> Inputs/Statusword @bit 8
//     Drive/Inputs/In/nState4 @bit 1 <-> WcState/InputToggle
//     Drive/Inputs/In/nState4 <-> WcState/WcState
//     Drive/Outputs/Out/nCtrl1 <-> Outputs/Controlword
//     Drive/Outputs/Out/nCtrl2 <-> Outputs/Controlword @bit 8
//     Drive/Outputs/Out/nDataOut1 <-> Outputs/Target position
//     Enc/Inputs/In/nDataIn1 <-> Inputs/Position actual value
//     Enc/Inputs/In/nDataIn3 <-> Inputs/Touch probe pos1 pos value
//     Enc/Inputs/In/nDataIn5 <-> Inputs/Touch probe pos2 pos value
//     Enc/Inputs/In/nDcInputTime <-> InfoData/DcInputShift
//     Enc/Inputs/In/nState4 @bit 1 <-> WcState/InputToggle
//     Enc/Inputs/In/nState4 <-> WcState/WcState
//     Enc/Inputs/In/nState5 <-> Inputs/Touch probe status
//     Enc/Inputs/In/nState6 <-> Inputs/Touch probe status @bit 8
//     Enc/Outputs/Out/nCtrl5 <-> Outputs/Touch probe function
//     Enc/Outputs/Out/nCtrl6 <-> Outputs/Touch probe function @bit 8
//   NC-Task 1 SAF/Axes/rem9_Lift1 <-> rem_wf/rem9_Lift1
//     Drive/Inputs/In/nDataIn1 <-> Inputs/Following error actual value
//     Drive/Inputs/In/nDataIn3[0] <-> Inputs/Torque actual value
//     Drive/Inputs/In/nDcOutputTime <-> InfoData/DcOutputShift
//     Drive/Inputs/In/nState1 <-> Inputs/Statusword
//     Drive/Inputs/In/nState2 <-> Inputs/Statusword @bit 8
//     Drive/Inputs/In/nState4 @bit 1 <-> WcState/InputToggle
//     Drive/Inputs/In/nState4 <-> WcState/WcState
//     Drive/Outputs/Out/nCtrl1 <-> Outputs/Controlword
//     Drive/Outputs/Out/nCtrl2 <-> Outputs/Controlword @bit 8
//     Drive/Outputs/Out/nDataOut1 <-> Outputs/Target position
//     Enc/Inputs/In/nDataIn1 <-> Inputs/Position actual value
//     Enc/Inputs/In/nDataIn3 <-> Inputs/Touch probe pos1 pos value
//     Enc/Inputs/In/nDataIn5 <-> Inputs/Touch probe pos2 pos value
//     Enc/Inputs/In/nDcInputTime <-> InfoData/DcInputShift
//     Enc/Inputs/In/nState4 @bit 1 <-> WcState/InputToggle
//     Enc/Inputs/In/nState4 <-> WcState/WcState
//     Enc/Inputs/In/nState5 <-> Inputs/Touch probe status
//     Enc/Inputs/In/nState6 <-> Inputs/Touch probe status @bit 8
//     Enc/Outputs/Out/nCtrl5 <-> Outputs/Touch probe function
//     Enc/Outputs/Out/nCtrl6 <-> Outputs/Touch probe function @bit 8
//   kittingDeca/kittingDeca Instance <-> pm side/fr0_dio
//     PlcTask Inputs/G_IO.arDI[75]/Ch[0] <-> Module 1 (GL20-1600END)/1600END input-bit maping/Digital input CH1-bit0
//     PlcTask Inputs/G_IO.arDI[75]/Ch[10] <-> Module 1 (GL20-1600END)/1600END input-bit maping/Digital input CH2-bit2
//     PlcTask Inputs/G_IO.arDI[75]/Ch[11] <-> Module 1 (GL20-1600END)/1600END input-bit maping/Digital input CH2-bit3
